LIN {X 0,Y 171.805,Z 482.478,A -85,B 0,C 180,E1 -24434.283,E2 -24434.283} C_VEL
LIN {X 0,Y 169.937,Z 475.539,A -85,B 0,C 180,E1 -24436.969,E2 -24436.969} C_VEL
LIN {X 0,Y 167.146,Z 467.963,A -85,B 0,C 180,E1 -24440.038,E2 -24440.038} C_VEL
LIN {X 0,Y 163.799,Z 461.064,A -85,B 0,C 180,E1 -24443.08,E2 -24443.08} C_VEL
LIN {X 0,Y 159.672,Z 454.191,A -85,B 0,C 180,E1 -24446.526,E2 -24446.526} C_VEL
LIN {X 0,Y 157.443,Z 450.927,A -85,B 0,C 180,E1 -24448.364,E2 -24448.364} C_VEL
LIN {X 0,Y 155.234,Z 452.338,A -85,B 0,C 180,E1 -24449.474,E2 -24449.474} C_VEL
LIN {X 0,Y 153.646,Z 452.709,A -85,B 0,C 180,E1 -24450.439,E2 -24450.439} C_VEL
LIN {X 0,Y 151.566,Z 454.907,A -85,B 0,C 180,E1 -24451.431,E2 -24451.431} C_VEL
LIN {X 0,Y 150.413,Z 455.475,A -85,B 0,C 180,E1 -24452.143,E2 -24452.143} C_VEL
LIN {X 0,Y 149.346,Z 455.04,A -85,B 0,C 180,E1 -24453.036,E2 -24453.036} C_VEL
LIN {X 0,Y 149.052,Z 454.259,A -85,B 0,C 180,E1 -24453.433,E2 -24453.433} C_VEL
LIN {X 0,Y 150.557,Z 461.284,A -85,B 0,C 180,E1 -24455.157,E2 -24455.157} C_VEL
LIN {X 0,Y 147.924,Z 476.238,A -85,B 0,C 180,E1 -24459.124,E2 -24459.124} C_VEL
LIN {X 0,Y 146.015,Z 488.722,A -85,B 0,C 180,E1 -24463.213,E2 -24463.213} C_VEL
LIN {X 0,Y 144.421,Z 500.063,A -85,B 0,C 180,E1 -24467.685,E2 -24467.685} C_VEL
LIN {X 0,Y 143.516,Z 508.412,A -85,B 0,C 180,E1 -24471.551,E2 -24471.551} C_VEL
LIN {X 0,Y 143,Z 518.672,A -85,B 0,C 180,E1 -24477.182,E2 -24477.182} C_VEL
LIN {X 0,Y 143.402,Z 525.259,A -85,B 0,C 180,E1 -24481.403,E2 -24481.403} C_VEL
LIN {X 0,Y 144.633,Z 532.666,A -85,B 0,C 180,E1 -24486.977,E2 -24486.977} C_VEL
LIN {X 0,Y 147.071,Z 538.788,A -85,B 0,C 180,E1 -24492.417,E2 -24492.417} C_VEL
LIN {X 0,Y 150.905,Z 543.761,A -85,B 0,C 180,E1 -24497.62,E2 -24497.62} C_VEL
LIN {X 0,Y 157.426,Z 548.456,A -85,B 0,C 180,E1 -24503.69,E2 -24503.69} C_VEL
LIN {X 0,Y 163.782,Z 551.125,A -85,B 0,C 180,E1 -24508.165,E2 -24508.165} C_VEL
LIN {X 0,Y 171.252,Z 552.834,A -85,B 0,C 180,E1 -24512.242,E2 -24512.242} C_VEL
LIN {X 0,Y 179.727,Z 553.572,A -85,B 0,C 180,E1 -24515.912,E2 -24515.912} C_VEL
LIN {X 0,Y 191.407,Z 553.206,A -85,B 0,C 180,E1 -24519.91,E2 -24519.91} C_VEL
LIN {X 0,Y 190.821,Z 553.718,A -85,B 0,C 180,E1 -24520.483,E2 -24520.483} C_VEL
LIN {X 0,Y 178.138,Z 559.175,A -85,B 0,C 180,E1 -24524.751,E2 -24524.751} C_VEL
LIN {X 0,Y 167.661,Z 563.079,A -85,B 0,C 180,E1 -24528.983,E2 -24528.983} C_VEL
LIN {X 0,Y 157.807,Z 566.417,A -85,B 0,C 180,E1 -24534.62,E2 -24534.62} C_VEL
LIN {X 0,Y 151.849,Z 568.111,A -85,B 0,C 180,E1 -24539.392,E2 -24539.392} C_VEL
LIN {X 0,Y 145.897,Z 569.336,A -85,B 0,C 180,E1 -24547.33,E2 -24547.33} C_VEL
LIN {X 0,Y 145.518,Z 569.56,A -85,B 0,C 180,E1 -24548.016,E2 -24548.016} C_VEL
LIN {X 0,Y 143.23,Z 574.219,A -85,B 0,C 180,E1 -24552.875,E2 -24552.875} C_VEL
LIN {X 0,Y 142.497,Z 576.289,A -85,B 0,C 180,E1 -24555.72,E2 -24555.72} C_VEL
LIN {X 0,Y 142.186,Z 579.073,A -85,B 0,C 180,E1 -24561.325,E2 -24561.325} C_VEL
LIN {X 0,Y 142.538,Z 579.938,A -85,B 0,C 180,E1 -24564.338,E2 -24564.338} C_VEL
LIN {X 0,Y 143.039,Z 580.34,A -85,B 0,C 180,E1 -24567.181,E2 -24567.181} C_VEL
LIN {X 0,Y 143.855,Z 580.307,A -85,B 0,C 180,E1 -24569.997,E2 -24569.997} C_VEL
LIN {X 0,Y 143.134,Z 579.601,A -85,B 0,C 180,E1 -24572.811,E2 -24572.811} C_VEL
LIN {X 0,Y 142.679,Z 578.492,A -85,B 0,C 180,E1 -24575.651,E2 -24575.651} C_VEL
LIN {X 0,Y 142.304,Z 576.622,A -85,B 0,C 180,E1 -24578.983,E2 -24578.983} C_VEL
LIN {X 0,Y 142.415,Z 572.404,A -85,B 0,C 180,E1 -24584.282,E2 -24584.282} C_VEL
LIN {X 0,Y 143.415,Z 567.754,A -85,B 0,C 180,E1 -24588.571,E2 -24588.571} C_VEL
LIN {X 0,Y 145.217,Z 561.884,A -85,B 0,C 180,E1 -24592.775,E2 -24592.775} C_VEL
LIN {X 0,Y 147.915,Z 554.582,A -85,B 0,C 180,E1 -24596.829,E2 -24596.829} C_VEL
LIN {X 0,Y 151.265,Z 545.507,A -85,B 0,C 180,E1 -24600.732,E2 -24600.732} C_VEL
LIN {X 0,Y 152.321,Z 541.956,A -85,B 0,C 180,E1 -24602.042,E2 -24602.042} C_VEL
LIN {X 0,Y 153.79,Z 532.793,A -85,B 0,C 180,E1 -24605.167,E2 -24605.167} C_VEL
LIN {X 0,Y 155.409,Z 522.571,A -85,B 0,C 180,E1 -24608.032,E2 -24608.032} C_VEL
LIN {X 0,Y 156.504,Z 514.859,A -85,B 0,C 180,E1 -24609.836,E2 -24609.836} C_VEL
LIN {X 0,Y 156.689,Z 509.881,A -85,B 0,C 180,E1 -24610.999,E2 -24610.999} C_VEL
LIN {X 0,Y 155.545,Z 501.863,A -85,B 0,C 180,E1 -24613.085,E2 -24613.085} C_VEL
LIN {X 0,Y 154.315,Z 495.338,A -85,B 0,C 180,E1 -24614.705,E2 -24614.705} C_VEL
LIN {X 0,Y 153.628,Z 488.352,A -85,B 0,C 180,E1 -24616.066,E2 -24616.066} C_VEL
LIN {X 0,Y 152.596,Z 475.837,A -85,B 0,C 180,E1 -24618.1,E2 -24618.1} C_VEL
LIN {X 0,Y 151.177,Z 468.093,A -85,B 0,C 180,E1 -24619.396,E2 -24619.396} C_VEL
LIN {X 0,Y 145.37,Z 455.802,A -85,B 0,C 180,E1 -24622.894,E2 -24622.894} C_VEL
LIN {X 0,Y 144.25,Z 450.728,A -85,B 0,C 180,E1 -24625.337,E2 -24625.337} C_VEL
LIN {X 0,Y 142.137,Z 443.856,A -85,B 0,C 180,E1 -24629.227,E2 -24629.227} C_VEL
LIN {X 0,Y 140.598,Z 440.661,A -85,B 0,C 180,E1 -24631.65,E2 -24631.65} C_VEL
LIN {X 0,Y 139.499,Z 439.298,A -85,B 0,C 180,E1 -24633.037,E2 -24633.037} C_VEL
LIN {X 0,Y 137.889,Z 436.001,A -85,B 0,C 180,E1 -24635.937,E2 -24635.937} C_VEL
LIN {X 0,Y 136.434,Z 433.163,A -85,B 0,C 180,E1 -24638.865,E2 -24638.865} C_VEL
LIN {X 0,Y 136.27,Z 432.124,A -85,B 0,C 180,E1 -24639.825,E2 -24639.825} C_VEL
LIN {X 0,Y 136.489,Z 432.104,A -85,B 0,C 180,E1 -24648.115,E2 -24648.115} C_VEL
LIN {X 0,Y 136.58,Z 432.088,A -85,B 0,C 180,E1 -24651.12,E2 -24651.12} C_VEL
LIN {X 0,Y 137.127,Z 432.018,A -85,B 0,C 180,E1 -24660.001,E2 -24660.001} C_VEL
LIN {X 0,Y 136.571,Z 432.045,A -85,B 0,C 180,E1 -24668.882,E2 -24668.882} C_VEL
LIN {X 0,Y 136.483,Z 432.078,A -85,B 0,C 180,E1 -24671.956,E2 -24671.956} C_VEL
LIN {X 0,Y 136.244,Z 432.129,A -85,B 0,C 180,E1 -24678.03,E2 -24678.03} C_VEL
LIN {X 0,Y 136.191,Z 432.134,A -85,B 0,C 180,E1 -24681.751,E2 -24681.751} C_VEL
LIN {X 0,Y 136.093,Z 432.113,A -85,B 0,C 180,E1 -24688.618,E2 -24688.618} C_VEL
LIN {X 0,Y 136.142,Z 432.245,A -85,B 0,C 180,E1 -24692.385,E2 -24692.385} C_VEL
LIN {X 0,Y 137.183,Z 435.226,A -85,B 0,C 180,E1 -24695.757,E2 -24695.757} C_VEL
LIN {X 0,Y 141.142,Z 440.004,A -85,B 0,C 180,E1 -24698.55,E2 -24698.55} C_VEL
LIN {X 0,Y 144.042,Z 443.761,A -85,B 0,C 180,E1 -24700.508,E2 -24700.508} C_VEL
LIN {X 0,Y 146.952,Z 448.113,A -85,B 0,C 180,E1 -24702.496,E2 -24702.496} C_VEL
LIN {X 0,Y 150.969,Z 454.759,A -85,B 0,C 180,E1 -24705.307,E2 -24705.307} C_VEL
LIN {X 0,Y 155.269,Z 463.772,A -85,B 0,C 180,E1 -24708.703,E2 -24708.703} C_VEL
LIN {X 0,Y 158.22,Z 471.79,A -85,B 0,C 180,E1 -24711.551,E2 -24711.551} C_VEL
LIN {X 0,Y 160.626,Z 481.017,A -85,B 0,C 180,E1 -24714.765,E2 -24714.765} C_VEL
LIN {X 0,Y 160.992,Z 482.859,A -85,B 0,C 180,E1 -24715.427,E2 -24715.427} C_VEL
LIN {X 0,Y 160.557,Z 485.505,A -85,B 0,C 180,E1 -24716.08,E2 -24716.08} C_VEL
LIN {X 0,Y 156.85,Z 496.328,A -85,B 0,C 180,E1 -24718.75,E2 -24718.75} C_VEL
LIN {X 0,Y 152.896,Z 506.216,A -85,B 0,C 180,E1 -24721.895,E2 -24721.895} C_VEL
LIN {X 0,Y 148.976,Z 515.07,A -85,B 0,C 180,E1 -24725.624,E2 -24725.624} C_VEL
LIN {X 0,Y 145.507,Z 522.195,A -85,B 0,C 180,E1 -24729.505,E2 -24729.505} C_VEL
LIN {X 0,Y 143.222,Z 526.998,A -85,B 0,C 180,E1 -24732.88,E2 -24732.88} C_VEL
LIN {X 0,Y 140.788,Z 531.675,A -85,B 0,C 180,E1 -24737.022,E2 -24737.022} C_VEL
LIN {X 0,Y 138.855,Z 535.27,A -85,B 0,C 180,E1 -24741.27,E2 -24741.27} C_VEL
LIN {X 0,Y 137.973,Z 537.117,A -85,B 0,C 180,E1 -24744.156,E2 -24744.156} C_VEL
LIN {X 0,Y 137.419,Z 538.522,A -85,B 0,C 180,E1 -24747.072,E2 -24747.072} C_VEL
LIN {X 0,Y 137.226,Z 540.113,A -85,B 0,C 180,E1 -24752.939,E2 -24752.939} C_VEL
LIN {X 0,Y 137.317,Z 540.381,A -85,B 0,C 180,E1 -24755.878,E2 -24755.878} C_VEL
LIN {X 0,Y 137.608,Z 540.235,A -85,B 0,C 180,E1 -24758.817,E2 -24758.817} C_VEL
LIN {X 0,Y 139.808,Z 538.683,A -85,B 0,C 180,E1 -24764.56,E2 -24764.56} C_VEL
LIN {X 0,Y 141.286,Z 537.324,A -85,B 0,C 180,E1 -24767.368,E2 -24767.368} C_VEL
LIN {X 0,Y 143.838,Z 534.273,A -85,B 0,C 180,E1 -24771.819,E2 -24771.819} C_VEL
LIN {X 0,Y 147.707,Z 529.137,A -85,B 0,C 180,E1 -24776.876,E2 -24776.876} C_VEL
LIN {X 0,Y 151.298,Z 523.764,A -85,B 0,C 180,E1 -24780.731,E2 -24780.731} C_VEL
LIN {X 0,Y 155.503,Z 516.959,A -85,B 0,C 180,E1 -24784.401,E2 -24784.401} C_VEL
LIN {X 0,Y 160.227,Z 508.406,A -85,B 0,C 180,E1 -24787.888,E2 -24787.888} C_VEL
LIN {X 0,Y 164.531,Z 499.594,A -85,B 0,C 180,E1 -24790.651,E2 -24790.651} C_VEL
LIN {X 0,Y 167.149,Z 493.293,A -85,B 0,C 180,E1 -24792.282,E2 -24792.282} C_VEL
LIN {X 0,Y 166.758,Z 488.389,A -85,B 0,C 180,E1 -24794.236,E2 -24794.236} C_VEL
LIN {X 0,Y 164.998,Z 480.301,A -85,B 0,C 180,E1 -24797.615,E2 -24797.615} C_VEL
LIN {X 0,Y 162.856,Z 473.543,A -85,B 0,C 180,E1 -24800.545,E2 -24800.545} C_VEL
LIN {X 0,Y 159.432,Z 465.725,A -85,B 0,C 180,E1 -24804.261,E2 -24804.261} C_VEL
LIN {X 0,Y 155.545,Z 458.948,A -85,B 0,C 180,E1 -24807.987,E2 -24807.987} C_VEL
LIN {X 0,Y 154.773,Z 458.892,A -85,B 0,C 180,E1 -24808.475,E2 -24808.475} C_VEL
LIN {X 0,Y 153.201,Z 459.625,A -85,B 0,C 180,E1 -24809.312,E2 -24809.312} C_VEL
LIN {X 0,Y 150.645,Z 461.659,A -85,B 0,C 180,E1 -24810.559,E2 -24810.559} C_VEL
LIN {X 0,Y 148.706,Z 462.303,A -85,B 0,C 180,E1 -24811.795,E2 -24811.795} C_VEL
LIN {X 0,Y 144.741,Z 465.331,A -85,B 0,C 180,E1 -24814.086,E2 -24814.086} C_VEL
LIN {X 0,Y 143.085,Z 466.026,A -85,B 0,C 180,E1 -24815.322,E2 -24815.322} C_VEL
LIN {X 0,Y 142.719,Z 465.473,A -85,B 0,C 180,E1 -24815.932,E2 -24815.932} C_VEL
LIN {X 0,Y 140.372,Z 478.948,A -85,B 0,C 180,E1 -24819.866,E2 -24819.866} C_VEL
LIN {X 0,Y 138.522,Z 491.22,A -85,B 0,C 180,E1 -24824.213,E2 -24824.213} C_VEL
LIN {X 0,Y 136.942,Z 503.88,A -85,B 0,C 180,E1 -24829.651,E2 -24829.651} C_VEL
LIN {X 0,Y 135.988,Z 515.026,A -85,B 0,C 180,E1 -24835.553,E2 -24835.553} C_VEL
LIN {X 0,Y 136.288,Z 523.292,A -85,B 0,C 180,E1 -24840.738,E2 -24840.738} C_VEL
LIN {X 0,Y 137.599,Z 532.127,A -85,B 0,C 180,E1 -24847.335,E2 -24847.335} C_VEL
LIN {X 0,Y 140.151,Z 538.583,A -85,B 0,C 180,E1 -24853.041,E2 -24853.041} C_VEL
LIN {X 0,Y 145.344,Z 545.059,A -85,B 0,C 180,E1 -24859.784,E2 -24859.784} C_VEL
LIN {X 0,Y 150.972,Z 549.028,A -85,B 0,C 180,E1 -24864.769,E2 -24864.769} C_VEL
LIN {X 0,Y 157.609,Z 552.021,A -85,B 0,C 180,E1 -24869.373,E2 -24869.373} C_VEL
LIN {X 0,Y 165.381,Z 554.072,A -85,B 0,C 180,E1 -24873.534,E2 -24873.534} C_VEL
LIN {X 0,Y 174.177,Z 555.197,A -85,B 0,C 180,E1 -24877.246,E2 -24877.246} C_VEL
LIN {X 0,Y 181.439,Z 555.419,A -85,B 0,C 180,E1 -24879.775,E2 -24879.775} C_VEL
LIN {X 0,Y 180.961,Z 555.879,A -85,B 0,C 180,E1 -24880.385,E2 -24880.385} C_VEL
LIN {X 0,Y 168.483,Z 560.407,A -85,B 0,C 180,E1 -24884.833,E2 -24884.833} C_VEL
LIN {X 0,Y 159.674,Z 563.108,A -85,B 0,C 180,E1 -24888.68,E2 -24888.68} C_VEL
LIN {X 0,Y 152.091,Z 565.208,A -85,B 0,C 180,E1 -24893.075,E2 -24893.075} C_VEL
LIN {X 0,Y 143.319,Z 567.038,A -85,B 0,C 180,E1 -24900.632,E2 -24900.632} C_VEL
LIN {X 0,Y 139.662,Z 567.468,A -85,B 0,C 180,E1 -24905.885,E2 -24905.885} C_VEL
LIN {X 0,Y 136.991,Z 572.091,A -85,B 0,C 180,E1 -24910.518,E2 -24910.518} C_VEL
LIN {X 0,Y 135.568,Z 575.311,A -85,B 0,C 180,E1 -24914.974,E2 -24914.974} C_VEL
LIN {X 0,Y 135.12,Z 576.919,A -85,B 0,C 180,E1 -24917.989,E2 -24917.989} C_VEL
LIN {X 0,Y 135.45,Z 578.932,A -85,B 0,C 180,E1 -24924.04,E2 -24924.04} C_VEL
LIN {X 0,Y 135.939,Z 579.326,A -85,B 0,C 180,E1 -24927.033,E2 -24927.033} C_VEL
LIN {X 0,Y 136.764,Z 579.281,A -85,B 0,C 180,E1 -24929.997,E2 -24929.997} C_VEL
LIN {X 0,Y 136.03,Z 578.564,A -85,B 0,C 180,E1 -24932.958,E2 -24932.958} C_VEL
LIN {X 0,Y 135.579,Z 577.444,A -85,B 0,C 180,E1 -24935.947,E2 -24935.947} C_VEL
LIN {X 0,Y 135.24,Z 575.771,A -85,B 0,C 180,E1 -24939.118,E2 -24939.118} C_VEL
LIN {X 0,Y 135.425,Z 571.309,A -85,B 0,C 180,E1 -24945.036,E2 -24945.036} C_VEL
LIN {X 0,Y 136.585,Z 566.64,A -85,B 0,C 180,E1 -24949.536,E2 -24949.536} C_VEL
LIN {X 0,Y 138.827,Z 560.132,A -85,B 0,C 180,E1 -24954.325,E2 -24954.325} C_VEL
LIN {X 0,Y 142.076,Z 552.029,A -85,B 0,C 180,E1 -24958.832,E2 -24958.832} C_VEL
LIN {X 0,Y 145.122,Z 544.318,A -85,B 0,C 180,E1 -24962.185,E2 -24962.185} C_VEL
LIN {X 0,Y 147.098,Z 534.44,A -85,B 0,C 180,E1 -24965.904,E2 -24965.904} C_VEL
LIN {X 0,Y 149.05,Z 523.917,A -85,B 0,C 180,E1 -24969.094,E2 -24969.094} C_VEL
LIN {X 0,Y 150.937,Z 512.662,A -85,B 0,C 180,E1 -24971.842,E2 -24971.842} C_VEL
LIN {X 0,Y 152.621,Z 501.143,A -85,B 0,C 180,E1 -24974.056,E2 -24974.056} C_VEL
LIN {X 0,Y 153.683,Z 490.333,A -85,B 0,C 180,E1 -24975.732,E2 -24975.732} C_VEL
LIN {X 0,Y 153.628,Z 488.352,A -85,B 0,C 180,E1 -24976.066,E2 -24976.066} C_VEL
LIN {X 0,Y 152.956,Z 483.098,A -85,B 0,C 180,E1 -24977.077,E2 -24977.077} C_VEL
LIN {X 0,Y 150.674,Z 476.845,A -85,B 0,C 180,E1 -24978.733,E2 -24978.733} C_VEL
LIN {X 0,Y 146.728,Z 469.819,A -85,B 0,C 180,E1 -24981.137,E2 -24981.137} C_VEL
LIN {X 0,Y 143.421,Z 464.323,A -85,B 0,C 180,E1 -24983.156,E2 -24983.156} C_VEL
LIN {X 0,Y 138.725,Z 454.306,A -85,B 0,C 180,E1 -24986.569,E2 -24986.569} C_VEL
LIN {X 0,Y 137.507,Z 449.61,A -85,B 0,C 180,E1 -24989.264,E2 -24989.264} C_VEL
LIN {X 0,Y 135.708,Z 445.682,A -85,B 0,C 180,E1 -24992.22,E2 -24992.22} C_VEL
LIN {X 0,Y 131.769,Z 438.096,A -85,B 0,C 180,E1 -24999.716,E2 -24999.716} C_VEL
LIN {X 0,Y 129.406,Z 433.796,A -85,B 0,C 180,E1 -25005.855,E2 -25005.855} C_VEL
LIN {X 0,Y 129.333,Z 432.999,A -85,B 0,C 180,E1 -25007.048,E2 -25007.048} C_VEL
LIN {X 0,Y 129.506,Z 432.966,A -85,B 0,C 180,E1 -25010.631,E2 -25010.631} C_VEL
LIN {X 0,Y 130.082,Z 432.895,A -85,B 0,C 180,E1 -25020.001,E2 -25020.001} C_VEL
LIN {X 0,Y 129.5,Z 432.924,A -85,B 0,C 180,E1 -25029.371,E2 -25029.371} C_VEL
LIN {X 0,Y 129.386,Z 432.969,A -85,B 0,C 180,E1 -25032.55,E2 -25032.55} C_VEL
LIN {X 0,Y 129.153,Z 433.019,A -85,B 0,C 180,E1 -25039.057,E2 -25039.057} C_VEL
LIN {X 0,Y 129.013,Z 433.04,A -85,B 0,C 180,E1 -25044.973,E2 -25044.973} C_VEL
LIN {X 0,Y 129.044,Z 433.273,A -85,B 0,C 180,E1 -25045.831,E2 -25045.831} C_VEL
LIN {X 0,Y 130.673,Z 436.736,A -85,B 0,C 180,E1 -25051.288,E2 -25051.288} C_VEL
LIN {X 0,Y 136.497,Z 443.699,A -85,B 0,C 180,E1 -25056.194,E2 -25056.194} C_VEL
LIN {X 0,Y 140.572,Z 449.281,A -85,B 0,C 180,E1 -25059.371,E2 -25059.371} C_VEL
LIN {X 0,Y 145.033,Z 456.594,A -85,B 0,C 180,E1 -25062.916,E2 -25062.916} C_VEL
LIN {X 0,Y 149.652,Z 466.342,A -85,B 0,C 180,E1 -25067.014,E2 -25067.014} C_VEL
LIN {X 0,Y 152.721,Z 475.183,A -85,B 0,C 180,E1 -25070.428,E2 -25070.428} C_VEL
LIN {X 0,Y 154.852,Z 484.253,A -85,B 0,C 180,E1 -25073.846,E2 -25073.846} C_VEL
LIN {X 0,Y 155.065,Z 485.477,A -85,B 0,C 180,E1 -25074.305,E2 -25074.305} C_VEL
LIN {X 0,Y 151.601,Z 495.729,A -85,B 0,C 180,E1 -25076.838,E2 -25076.838} C_VEL
LIN {X 0,Y 147.528,Z 505.678,A -85,B 0,C 180,E1 -25079.99,E2 -25079.99} C_VEL
LIN {X 0,Y 143.224,Z 514.916,A -85,B 0,C 180,E1 -25083.796,E2 -25083.796} C_VEL
LIN {X 0,Y 139.531,Z 522.236,A -85,B 0,C 180,E1 -25087.808,E2 -25087.808} C_VEL
LIN {X 0,Y 136.539,Z 528.097,A -85,B 0,C 180,E1 -25092.015,E2 -25092.015} C_VEL
LIN {X 0,Y 133.953,Z 532.756,A -85,B 0,C 180,E1 -25096.347,E2 -25096.347} C_VEL
LIN {X 0,Y 131.917,Z 536.331,A -85,B 0,C 180,E1 -25100.807,E2 -25100.807} C_VEL
LIN {X 0,Y 130.987,Z 538.169,A -85,B 0,C 180,E1 -25103.843,E2 -25103.843} C_VEL
LIN {X 0,Y 130.402,Z 539.557,A -85,B 0,C 180,E1 -25106.914,E2 -25106.914} C_VEL
LIN {X 0,Y 130.206,Z 541.131,A -85,B 0,C 180,E1 -25113.097,E2 -25113.097} C_VEL
LIN {X 0,Y 130.324,Z 541.387,A -85,B 0,C 180,E1 -25116.195,E2 -25116.195} C_VEL
LIN {X 0,Y 130.661,Z 541.227,A -85,B 0,C 180,E1 -25119.289,E2 -25119.289} C_VEL
LIN {X 0,Y 133.016,Z 539.656,A -85,B 0,C 180,E1 -25125.321,E2 -25125.321} C_VEL
LIN {X 0,Y 134.591,Z 538.281,A -85,B 0,C 180,E1 -25128.262,E2 -25128.262} C_VEL
LIN {X 0,Y 137.314,Z 535.23,A -85,B 0,C 180,E1 -25132.884,E2 -25132.884} C_VEL
LIN {X 0,Y 141.464,Z 530.053,A -85,B 0,C 180,E1 -25138.165,E2 -25138.165} C_VEL
LIN {X 0,Y 145.292,Z 524.656,A -85,B 0,C 180,E1 -25142.15,E2 -25142.15} C_VEL
LIN {X 0,Y 149.739,Z 517.814,A -85,B 0,C 180,E1 -25145.925,E2 -25145.925} C_VEL
LIN {X 0,Y 154.739,Z 509.226,A -85,B 0,C 180,E1 -25149.487,E2 -25149.487} C_VEL
LIN {X 0,Y 159.252,Z 500.377,A -85,B 0,C 180,E1 -25152.302,E2 -25152.302} C_VEL
LIN {X 0,Y 161.44,Z 495.179,A -85,B 0,C 180,E1 -25153.72,E2 -25153.72} C_VEL
LIN {X 0,Y 160.715,Z 489.007,A -85,B 0,C 180,E1 -25156.469,E2 -25156.469} C_VEL
LIN {X 0,Y 159.299,Z 482.369,A -85,B 0,C 180,E1 -25159.484,E2 -25159.484} C_VEL
LIN {X 0,Y 156.998,Z 475.117,A -85,B 0,C 180,E1 -25162.98,E2 -25162.98} C_VEL
LIN {X 0,Y 154.432,Z 469.217,A -85,B 0,C 180,E1 -25166.117,E2 -25166.117} C_VEL
LIN {X 0,Y 152.726,Z 466,A -85,B 0,C 180,E1 -25168.048,E2 -25168.048} C_VEL
LIN {X 0,Y 150.464,Z 467.627,A -85,B 0,C 180,E1 -25169.082,E2 -25169.082} C_VEL
LIN {X 0,Y 146.504,Z 469.484,A -85,B 0,C 180,E1 -25171.332,E2 -25171.332} C_VEL
LIN {X 0,Y 144.368,Z 471.091,A -85,B 0,C 180,E1 -25172.452,E2 -25172.452} C_VEL
LIN {X 0,Y 142.493,Z 472.128,A -85,B 0,C 180,E1 -25173.646,E2 -25173.646} C_VEL
LIN {X 0,Y 140.43,Z 473.854,A -85,B 0,C 180,E1 -25174.825,E2 -25174.825} C_VEL
LIN {X 0,Y 136.879,Z 477.797,A -85,B 0,C 180,E1 -25176.551,E2 -25176.551} C_VEL
LIN {X 0,Y 135.859,Z 478.73,A -85,B 0,C 180,E1 -25177.171,E2 -25177.171} C_VEL
LIN {X 0,Y 134.15,Z 479.926,A -85,B 0,C 180,E1 -25178.485,E2 -25178.485} C_VEL
LIN {X 0,Y 133.163,Z 479.611,A -85,B 0,C 180,E1 -25180.037,E2 -25180.037} C_VEL
LIN {X 0,Y 131.339,Z 491.547,A -85,B 0,C 180,E1 -25184.48,E2 -25184.48} C_VEL
LIN {X 0,Y 129.85,Z 503.51,A -85,B 0,C 180,E1 -25189.868,E2 -25189.868} C_VEL
LIN {X 0,Y 128.926,Z 514.916,A -85,B 0,C 180,E1 -25196.092,E2 -25196.092} C_VEL
LIN {X 0,Y 129.318,Z 523.345,A -85,B 0,C 180,E1 -25201.556,E2 -25201.556} C_VEL
LIN {X 0,Y 130.607,Z 531.449,A -85,B 0,C 180,E1 -25207.73,E2 -25207.73} C_VEL
LIN {X 0,Y 133.254,Z 538.245,A -85,B 0,C 180,E1 -25213.729,E2 -25213.729} C_VEL
LIN {X 0,Y 137.462,Z 543.88,A -85,B 0,C 180,E1 -25219.409,E2 -25219.409} C_VEL
LIN {X 0,Y 144.565,Z 549.414,A -85,B 0,C 180,E1 -25225.946,E2 -25225.946} C_VEL
LIN {X 0,Y 151.513,Z 552.792,A -85,B 0,C 180,E1 -25230.679,E2 -25230.679} C_VEL
LIN {X 0,Y 159.592,Z 555.197,A -85,B 0,C 180,E1 -25234.923,E2 -25234.923} C_VEL
LIN {X 0,Y 170.706,Z 556.893,A -85,B 0,C 180,E1 -25239.38,E2 -25239.38} C_VEL
LIN {X 0,Y 171.241,Z 557.378,A -85,B 0,C 180,E1 -25240.306,E2 -25240.306} C_VEL
LIN {X 0,Y 158.865,Z 560.943,A -85,B 0,C 180,E1 -25244.939,E2 -25244.939} C_VEL
LIN {X 0,Y 150.328,Z 563.031,A -85,B 0,C 180,E1 -25249.114,E2 -25249.114} C_VEL
LIN {X 0,Y 139.976,Z 564.935,A -85,B 0,C 180,E1 -25256.472,E2 -25256.472} C_VEL
LIN {X 0,Y 133.887,Z 565.494,A -85,B 0,C 180,E1 -25263.744,E2 -25263.744} C_VEL
LIN {X 0,Y 131.038,Z 569.819,A -85,B 0,C 180,E1 -25267.946,E2 -25267.946} C_VEL
LIN {X 0,Y 129.082,Z 573.353,A -85,B 0,C 180,E1 -25272.572,E2 -25272.572} C_VEL
LIN {X 0,Y 128.121,Z 575.923,A -85,B 0,C 180,E1 -25277.322,E2 -25277.322} C_VEL
LIN {X 0,Y 128.359,Z 577.925,A -85,B 0,C 180,E1 -25283.71,E2 -25283.71} C_VEL
LIN {X 0,Y 128.838,Z 578.31,A -85,B 0,C 180,E1 -25286.87,E2 -25286.87} C_VEL
LIN {X 0,Y 129.676,Z 578.256,A -85,B 0,C 180,E1 -25289.997,E2 -25289.997} C_VEL
LIN {X 0,Y 128.927,Z 577.527,A -85,B 0,C 180,E1 -25293.121,E2 -25293.121} C_VEL
LIN {X 0,Y 128.463,Z 576.393,A -85,B 0,C 180,E1 -25296.278,E2 -25296.278} C_VEL
LIN {X 0,Y 128.082,Z 573.815,A -85,B 0,C 180,E1 -25301.069,E2 -25301.069} C_VEL
LIN {X 0,Y 128.474,Z 570.216,A -85,B 0,C 180,E1 -25305.87,E2 -25305.87} C_VEL
LIN {X 0,Y 129.811,Z 565.529,A -85,B 0,C 180,E1 -25310.6,E2 -25310.6} C_VEL
LIN {X 0,Y 132.512,Z 558.474,A -85,B 0,C 180,E1 -25315.944,E2 -25315.944} C_VEL
LIN {X 0,Y 135.806,Z 550.865,A -85,B 0,C 180,E1 -25320.298,E2 -25320.298} C_VEL
LIN {X 0,Y 138.886,Z 543.09,A -85,B 0,C 180,E1 -25323.819,E2 -25323.819} C_VEL
LIN {X 0,Y 140.987,Z 533.364,A -85,B 0,C 180,E1 -25327.632,E2 -25327.632} C_VEL
LIN {X 0,Y 143.273,Z 522.572,A -85,B 0,C 180,E1 -25330.997,E2 -25330.997} C_VEL
LIN {X 0,Y 145.434,Z 511.097,A -85,B 0,C 180,E1 -25333.861,E2 -25333.861} C_VEL
LIN {X 0,Y 147.465,Z 498.539,A -85,B 0,C 180,E1 -25336.28,E2 -25336.28} C_VEL
LIN {X 0,Y 148.217,Z 491.08,A -85,B 0,C 180,E1 -25337.493,E2 -25337.493} C_VEL
LIN {X 0,Y 147.659,Z 479.337,A -85,B 0,C 180,E1 -25339.595,E2 -25339.595} C_VEL
LIN {X 0,Y 146.686,Z 471.856,A -85,B 0,C 180,E1 -25340.931,E2 -25340.931} C_VEL
LIN {X 0,Y 143.421,Z 464.323,A -85,B 0,C 180,E1 -25343.156,E2 -25343.156} C_VEL
LIN {X 0,Y 140.911,Z 460.619,A -85,B 0,C 180,E1 -25344.732,E2 -25344.732} C_VEL
LIN {X 0,Y 136.291,Z 455.849,A -85,B 0,C 180,E1 -25347.787,E2 -25347.787} C_VEL
LIN {X 0,Y 131.421,Z 451.317,A -85,B 0,C 180,E1 -25352.093,E2 -25352.093} C_VEL
LIN {X 0,Y 130.236,Z 449.835,A -85,B 0,C 180,E1 -25353.644,E2 -25353.644} C_VEL
LIN {X 0,Y 126.937,Z 443.072,A -85,B 0,C 180,E1 -25360.599,E2 -25360.599} C_VEL
LIN {X 0,Y 124.67,Z 438.557,A -85,B 0,C 180,E1 -25366.969,E2 -25366.969} C_VEL
LIN {X 0,Y 122.838,Z 433.805,A -85,B 0,C 180,E1 -25378.771,E2 -25378.771} C_VEL
LIN {X 0,Y 123.036,Z 433.772,A -85,B 0,C 180,E1 -25380.001,E2 -25380.001} C_VEL
LIN {X 0,Y 122.404,Z 433.814,A -85,B 0,C 180,E1 -25387.137,E2 -25387.137} C_VEL
LIN {X 0,Y 122.355,Z 433.84,A -85,B 0,C 180,E1 -25392.473,E2 -25392.473} C_VEL
LIN {X 0,Y 122.802,Z 436.27,A -85,B 0,C 180,E1 -25400.084,E2 -25400.084} C_VEL
LIN {X 0,Y 124.245,Z 438.461,A -85,B 0,C 180,E1 -25405.581,E2 -25405.581} C_VEL
LIN {X 0,Y 127.692,Z 442.456,A -85,B 0,C 180,E1 -25409.467,E2 -25409.467} C_VEL
LIN {X 0,Y 129.418,Z 444.245,A -85,B 0,C 180,E1 -25411.175,E2 -25411.175} C_VEL
LIN {X 0,Y 133.877,Z 450.1,A -85,B 0,C 180,E1 -25415.388,E2 -25415.388} C_VEL
LIN {X 0,Y 137.193,Z 455.092,A -85,B 0,C 180,E1 -25418.4,E2 -25418.4} C_VEL
LIN {X 0,Y 140.314,Z 460.669,A -85,B 0,C 180,E1 -25421.301,E2 -25421.301} C_VEL
LIN {X 0,Y 143.701,Z 467.997,A -85,B 0,C 180,E1 -25424.743,E2 -25424.743} C_VEL
LIN {X 0,Y 146.466,Z 475.686,A -85,B 0,C 180,E1 -25428.051,E2 -25428.051} C_VEL
LIN {X 0,Y 148.475,Z 484.061,A -85,B 0,C 180,E1 -25431.455,E2 -25431.455} C_VEL
LIN {X 0,Y 149.139,Z 488.055,A -85,B 0,C 180,E1 -25433.076,E2 -25433.076} C_VEL
LIN {X 0,Y 145.198,Z 498.43,A -85,B 0,C 180,E1 -25435.775,E2 -25435.775} C_VEL
LIN {X 0,Y 140.682,Z 508.587,A -85,B 0,C 180,E1 -25439.203,E2 -25439.203} C_VEL
LIN {X 0,Y 136.333,Z 517.361,A -85,B 0,C 180,E1 -25443.192,E2 -25443.192} C_VEL
LIN {X 0,Y 132.503,Z 524.431,A -85,B 0,C 180,E1 -25447.388,E2 -25447.388} C_VEL
LIN {X 0,Y 129.889,Z 529.196,A -85,B 0,C 180,E1 -25451.06,E2 -25451.06} C_VEL
LIN {X 0,Y 127.166,Z 533.832,A -85,B 0,C 180,E1 -25455.603,E2 -25455.603} C_VEL
LIN {X 0,Y 124.988,Z 537.392,A -85,B 0,C 180,E1 -25460.292,E2 -25460.292} C_VEL
LIN {X 0,Y 124.006,Z 539.221,A -85,B 0,C 180,E1 -25463.495,E2 -25463.495} C_VEL
LIN {X 0,Y 123.387,Z 540.591,A -85,B 0,C 180,E1 -25466.738,E2 -25466.738} C_VEL
LIN {X 0,Y 123.188,Z 542.148,A -85,B 0,C 180,E1 -25473.274,E2 -25473.274} C_VEL
LIN {X 0,Y 123.336,Z 542.391,A -85,B 0,C 180,E1 -25476.547,E2 -25476.547} C_VEL
LIN {X 0,Y 123.724,Z 542.219,A -85,B 0,C 180,E1 -25479.815,E2 -25479.815} C_VEL
LIN {X 0,Y 126.249,Z 540.63,A -85,B 0,C 180,E1 -25486.164,E2 -25486.164} C_VEL
LIN {X 0,Y 127.932,Z 539.236,A -85,B 0,C 180,E1 -25489.249,E2 -25489.249} C_VEL
LIN {X 0,Y 130.853,Z 536.178,A -85,B 0,C 180,E1 -25494.067,E2 -25494.067} C_VEL
LIN {X 0,Y 134.052,Z 532.513,A -85,B 0,C 180,E1 -25498.158,E2 -25498.158} C_VEL
LIN {X 0,Y 137.925,Z 527.488,A -85,B 0,C 180,E1 -25502.349,E2 -25502.349} C_VEL
LIN {X 0,Y 142.511,Z 521.112,A -85,B 0,C 180,E1 -25506.287,E2 -25506.287} C_VEL
LIN {X 0,Y 146.802,Z 514.365,A -85,B 0,C 180,E1 -25509.518,E2 -25509.518} C_VEL
LIN {X 0,Y 151.267,Z 506.685,A -85,B 0,C 180,E1 -25512.355,E2 -25512.355} C_VEL
LIN {X 0,Y 155.502,Z 498.111,A -85,B 0,C 180,E1 -25514.91,E2 -25514.91} C_VEL
LIN {X 0,Y 155.678,Z 496.464,A -85,B 0,C 180,E1 -25515.595,E2 -25515.595} C_VEL
LIN {X 0,Y 154.577,Z 488.204,A -85,B 0,C 180,E1 -25519.616,E2 -25519.616} C_VEL
LIN {X 0,Y 152.784,Z 481.093,A -85,B 0,C 180,E1 -25523.273,E2 -25523.273} C_VEL
LIN {X 0,Y 150.388,Z 474.599,A -85,B 0,C 180,E1 -25526.935,E2 -25526.935} C_VEL
LIN {X 0,Y 149.941,Z 473.671,A -85,B 0,C 180,E1 -25527.536,E2 -25527.536} C_VEL
LIN {X 0,Y 146.01,Z 475.351,A -85,B 0,C 180,E1 -25529.641,E2 -25529.641} C_VEL
LIN {X 0,Y 141.786,Z 477.908,A -85,B 0,C 180,E1 -25531.907,E2 -25531.907} C_VEL
LIN {X 0,Y 139.562,Z 479.673,A -85,B 0,C 180,E1 -25533.049,E2 -25533.049} C_VEL
LIN {X 0,Y 135.809,Z 483.289,A -85,B 0,C 180,E1 -25534.733,E2 -25534.733} C_VEL
LIN {X 0,Y 134.715,Z 484.217,A -85,B 0,C 180,E1 -25535.331,E2 -25535.331} C_VEL
LIN {X 0,Y 132.835,Z 485.492,A -85,B 0,C 180,E1 -25536.62,E2 -25536.62} C_VEL
LIN {X 0,Y 131.244,Z 486.298,A -85,B 0,C 180,E1 -25537.984,E2 -25537.984} C_VEL
LIN {X 0,Y 129.392,Z 487.778,A -85,B 0,C 180,E1 -25539.325,E2 -25539.325} C_VEL
LIN {X 0,Y 127.323,Z 489.737,A -85,B 0,C 180,E1 -25540.658,E2 -25540.658} C_VEL
LIN {X 0,Y 125.364,Z 491.284,A -85,B 0,C 180,E1 -25542.379,E2 -25542.379} C_VEL
LIN {X 0,Y 124.275,Z 491.532,A -85,B 0,C 180,E1 -25544.156,E2 -25544.156} C_VEL
LIN {X 0,Y 124.213,Z 491.312,A -85,B 0,C 180,E1 -25544.595,E2 -25544.595} C_VEL
LIN {X 0,Y 122.753,Z 503.048,A -85,B 0,C 180,E1 -25550.109,E2 -25550.109} C_VEL
LIN {X 0,Y 121.933,Z 513.288,A -85,B 0,C 180,E1 -25555.868,E2 -25555.868} C_VEL
LIN {X 0,Y 122.308,Z 522.085,A -85,B 0,C 180,E1 -25561.646,E2 -25561.646} C_VEL
LIN {X 0,Y 123.623,Z 530.548,A -85,B 0,C 180,E1 -25568.17,E2 -25568.17} C_VEL
LIN {X 0,Y 126.384,Z 537.68,A -85,B 0,C 180,E1 -25574.491,E2 -25574.491} C_VEL
LIN {X 0,Y 132.082,Z 544.995,A -85,B 0,C 180,E1 -25581.867,E2 -25581.867} C_VEL
LIN {X 0,Y 138.218,Z 549.642,A -85,B 0,C 180,E1 -25587.233,E2 -25587.233} C_VEL
LIN {X 0,Y 145.483,Z 553.345,A -85,B 0,C 180,E1 -25592.099,E2 -25592.099} C_VEL
LIN {X 0,Y 153.886,Z 556.157,A -85,B 0,C 180,E1 -25596.42,E2 -25596.42} C_VEL
LIN {X 0,Y 161.63,Z 557.746,A -85,B 0,C 180,E1 -25599.579,E2 -25599.579} C_VEL
LIN {X 0,Y 160.591,Z 558.362,A -85,B 0,C 180,E1 -25600.569,E2 -25600.569} C_VEL
LIN {X 0,Y 149.354,Z 560.838,A -85,B 0,C 180,E1 -25605.099,E2 -25605.099} C_VEL
LIN {X 0,Y 137.483,Z 562.787,A -85,B 0,C 180,E1 -25612.159,E2 -25612.159} C_VEL
LIN {X 0,Y 131.355,Z 563.304,A -85,B 0,C 180,E1 -25617.65,E2 -25617.65} C_VEL
LIN {X 0,Y 128.421,Z 563.39,A -85,B 0,C 180,E1 -25621.308,E2 -25621.308} C_VEL
LIN {X 0,Y 124.445,Z 568.862,A -85,B 0,C 180,E1 -25626.71,E2 -25626.71} C_VEL
LIN {X 0,Y 122.253,Z 572.373,A -85,B 0,C 180,E1 -25631.564,E2 -25631.564} C_VEL
LIN {X 0,Y 121.161,Z 574.931,A -85,B 0,C 180,E1 -25636.58,E2 -25636.58} C_VEL
LIN {X 0,Y 121.253,Z 576.915,A -85,B 0,C 180,E1 -25643.34,E2 -25643.34} C_VEL
LIN {X 0,Y 121.737,Z 577.292,A -85,B 0,C 180,E1 -25646.687,E2 -25646.687} C_VEL
LIN {X 0,Y 122.589,Z 577.231,A -85,B 0,C 180,E1 -25649.996,E2 -25649.996} C_VEL
LIN {X 0,Y 121.823,Z 576.49,A -85,B 0,C 180,E1 -25653.304,E2 -25653.304} C_VEL
LIN {X 0,Y 121.112,Z 574.049,A -85,B 0,C 180,E1 -25659.432,E2 -25659.432} C_VEL
LIN {X 0,Y 121.265,Z 570.45,A -85,B 0,C 180,E1 -25665.114,E2 -25665.114} C_VEL
LIN {X 0,Y 122.48,Z 566.116,A -85,B 0,C 180,E1 -25670.134,E2 -25670.134} C_VEL
LIN {X 0,Y 124.514,Z 560.862,A -85,B 0,C 180,E1 -25674.807,E2 -25674.807} C_VEL
LIN {X 0,Y 127.785,Z 553.721,A -85,B 0,C 180,E1 -25679.665,E2 -25679.665} C_VEL
LIN {X 0,Y 131.671,Z 545.232,A -85,B 0,C 180,E1 -25684.082,E2 -25684.082} C_VEL
LIN {X 0,Y 134.13,Z 535.779,A -85,B 0,C 180,E1 -25688.192,E2 -25688.192} C_VEL
LIN {X 0,Y 136.453,Z 526.31,A -85,B 0,C 180,E1 -25691.534,E2 -25691.534} C_VEL
LIN {X 0,Y 138.817,Z 515.851,A -85,B 0,C 180,E1 -25694.523,E2 -25694.523} C_VEL
LIN {X 0,Y 141.254,Z 503.879,A -85,B 0,C 180,E1 -25697.206,E2 -25697.206} C_VEL
LIN {X 0,Y 142.861,Z 493.351,A -85,B 0,C 180,E1 -25699.09,E2 -25699.09} C_VEL
LIN {X 0,Y 142.617,Z 480.759,A -85,B 0,C 180,E1 -25701.534,E2 -25701.534} C_VEL
LIN {X 0,Y 142.077,Z 475.494,A -85,B 0,C 180,E1 -25702.571,E2 -25702.571} C_VEL
LIN {X 0,Y 137.727,Z 464.887,A -85,B 0,C 180,E1 -25706.075,E2 -25706.075} C_VEL
LIN {X 0,Y 135.073,Z 459.093,A -85,B 0,C 180,E1 -25708.21,E2 -25708.21} C_VEL
LIN {X 0,Y 131.791,Z 452.821,A -85,B 0,C 180,E1 -25711.035,E2 -25711.035} C_VEL
LIN {X 0,Y 130.236,Z 449.835,A -85,B 0,C 180,E1 -25713.644,E2 -25713.644} C_VEL
LIN {X 0,Y 128.41,Z 448.075,A -85,B 0,C 180,E1 -25716.013,E2 -25716.013} C_VEL
LIN {X 0,Y 124.728,Z 446.589,A -85,B 0,C 180,E1 -25720.13,E2 -25720.13} C_VEL
LIN {X 0,Y 120.888,Z 445.177,A -85,B 0,C 180,E1 -25725.41,E2 -25725.41} C_VEL
LIN {X 0,Y 120.136,Z 444.329,A -85,B 0,C 180,E1 -25727.233,E2 -25727.233} C_VEL
LIN {X 0,Y 119.467,Z 442.895,A -85,B 0,C 180,E1 -25729.836,E2 -25729.836} C_VEL
LIN {X 0,Y 118.155,Z 438.914,A -85,B 0,C 180,E1 -25740.001,E2 -25740.001} C_VEL
LIN {X 0,Y 117.597,Z 439.026,A -85,B 0,C 180,E1 -25750.329,E2 -25750.329} C_VEL
LIN {X 0,Y 117.689,Z 439.604,A -85,B 0,C 180,E1 -25753.821,E2 -25753.821} C_VEL
LIN {X 0,Y 117.829,Z 440.691,A -85,B 0,C 180,E1 -25757.129,E2 -25757.129} C_VEL
LIN {X 0,Y 122.61,Z 445.268,A -85,B 0,C 180,E1 -25764.795,E2 -25764.795} C_VEL
LIN {X 0,Y 125.824,Z 449.119,A -85,B 0,C 180,E1 -25768.801,E2 -25768.801} C_VEL
LIN {X 0,Y 127.188,Z 450.892,A -85,B 0,C 180,E1 -25770.395,E2 -25770.395} C_VEL
LIN {X 0,Y 130.876,Z 456.184,A -85,B 0,C 180,E1 -25774.44,E2 -25774.44} C_VEL
LIN {X 0,Y 133.624,Z 460.865,A -85,B 0,C 180,E1 -25777.408,E2 -25777.408} C_VEL
LIN {X 0,Y 136.799,Z 467.172,A -85,B 0,C 180,E1 -25780.923,E2 -25780.923} C_VEL
LIN {X 0,Y 139.818,Z 474.824,A -85,B 0,C 180,E1 -25784.727,E2 -25784.727} C_VEL
LIN {X 0,Y 141.837,Z 482.021,A -85,B 0,C 180,E1 -25788.01,E2 -25788.01} C_VEL
LIN {X 0,Y 143.165,Z 489.424,A -85,B 0,C 180,E1 -25791.257,E2 -25791.257} C_VEL
LIN {X 0,Y 143.128,Z 490.568,A -85,B 0,C 180,E1 -25791.695,E2 -25791.695} C_VEL
LIN {X 0,Y 138.848,Z 501.107,A -85,B 0,C 180,E1 -25794.603,E2 -25794.603} C_VEL
LIN {X 0,Y 134.707,Z 509.767,A -85,B 0,C 180,E1 -25797.676,E2 -25797.676} C_VEL
LIN {X 0,Y 130.116,Z 518.505,A -85,B 0,C 180,E1 -25801.8,E2 -25801.8} C_VEL
LIN {X 0,Y 126.067,Z 525.55,A -85,B 0,C 180,E1 -25806.165,E2 -25806.165} C_VEL
LIN {X 0,Y 123.278,Z 530.295,A -85,B 0,C 180,E1 -25810.002,E2 -25810.002} C_VEL
LIN {X 0,Y 120.399,Z 534.909,A -85,B 0,C 180,E1 -25814.775,E2 -25814.775} C_VEL
LIN {X 0,Y 118.07,Z 538.454,A -85,B 0,C 180,E1 -25819.717,E2 -25819.717} C_VEL
LIN {X 0,Y 117.029,Z 540.271,A -85,B 0,C 180,E1 -25823.106,E2 -25823.106} C_VEL
LIN {X 0,Y 116.097,Z 542.584,A -85,B 0,C 180,E1 -25830.004,E2 -25830.004} C_VEL
LIN {X 0,Y 116.17,Z 543.166,A -85,B 0,C 180,E1 -25833.472,E2 -25833.472} C_VEL
LIN {X 0,Y 116.353,Z 543.393,A -85,B 0,C 180,E1 -25836.942,E2 -25836.942} C_VEL
LIN {X 0,Y 116.798,Z 543.211,A -85,B 0,C 180,E1 -25840.404,E2 -25840.404} C_VEL
LIN {X 0,Y 119.513,Z 541.603,A -85,B 0,C 180,E1 -25847.103,E2 -25847.103} C_VEL
LIN {X 0,Y 121.315,Z 540.191,A -85,B 0,C 180,E1 -25850.344,E2 -25850.344} C_VEL
LIN {X 0,Y 124.458,Z 537.122,A -85,B 0,C 180,E1 -25855.376,E2 -25855.376} C_VEL
LIN {X 0,Y 127.871,Z 533.432,A -85,B 0,C 180,E1 -25859.651,E2 -25859.651} C_VEL
LIN {X 0,Y 132.029,Z 528.382,A -85,B 0,C 180,E1 -25863.985,E2 -25863.985} C_VEL
LIN {X 0,Y 136.896,Z 521.981,A -85,B 0,C 180,E1 -25868.033,E2 -25868.033} C_VEL
LIN {X 0,Y 142.385,Z 513.672,A -85,B 0,C 180,E1 -25872.004,E2 -25872.004} C_VEL
LIN {X 0,Y 147.123,Z 505.727,A -85,B 0,C 180,E1 -25874.801,E2 -25874.801} C_VEL
LIN {X 0,Y 149.76,Z 500.56,A -85,B 0,C 180,E1 -25876.346,E2 -25876.346} C_VEL
LIN {X 0,Y 149.991,Z 499.133,A -85,B 0,C 180,E1 -25876.966,E2 -25876.966} C_VEL
LIN {X 0,Y 149.341,Z 492.158,A -85,B 0,C 180,E1 -25880.635,E2 -25880.635} C_VEL
LIN {X 0,Y 147.924,Z 485.362,A -85,B 0,C 180,E1 -25884.424,E2 -25884.424} C_VEL
LIN {X 0,Y 146.767,Z 481.511,A -85,B 0,C 180,E1 -25886.744,E2 -25886.744} C_VEL
LIN {X 0,Y 145.362,Z 481.064,A -85,B 0,C 180,E1 -25887.87,E2 -25887.87} C_VEL
LIN {X 0,Y 140.958,Z 483.462,A -85,B 0,C 180,E1 -25890.092,E2 -25890.092} C_VEL
LIN {X 0,Y 138.542,Z 485.24,A -85,B 0,C 180,E1 -25891.188,E2 -25891.188} C_VEL
LIN {X 0,Y 133.861,Z 489.202,A -85,B 0,C 180,E1 -25893.2,E2 -25893.2} C_VEL
LIN {X 0,Y 131.389,Z 490.863,A -85,B 0,C 180,E1 -25894.663,E2 -25894.663} C_VEL
LIN {X 0,Y 127.67,Z 493.062,A -85,B 0,C 180,E1 -25897.334,E2 -25897.334} C_VEL
LIN {X 0,Y 125.455,Z 494.95,A -85,B 0,C 180,E1 -25898.645,E2 -25898.645} C_VEL
LIN {X 0,Y 123.648,Z 496.26,A -85,B 0,C 180,E1 -25900.059,E2 -25900.059} C_VEL
LIN {X 0,Y 120.998,Z 497.67,A -85,B 0,C 180,E1 -25903.116,E2 -25903.116} C_VEL
LIN {X 0,Y 117.536,Z 500.876,A -85,B 0,C 180,E1 -25906.161,E2 -25906.161} C_VEL
LIN {X 0,Y 115.758,Z 502.032,A -85,B 0,C 180,E1 -25909.505,E2 -25909.505} C_VEL
LIN {X 0,Y 115.735,Z 502.056,A -85,B 0,C 180,E1 -25910.165,E2 -25910.165} C_VEL
LIN {X 0,Y 114.9,Z 512.912,A -85,B 0,C 180,E1 -25916.492,E2 -25916.492} C_VEL
LIN {X 0,Y 115.374,Z 521.88,A -85,B 0,C 180,E1 -25922.618,E2 -25922.618} C_VEL
LIN {X 0,Y 117.197,Z 531.479,A -85,B 0,C 180,E1 -25930.363,E2 -25930.363} C_VEL
LIN {X 0,Y 120.55,Z 538.664,A -85,B 0,C 180,E1 -25936.947,E2 -25936.947} C_VEL
LIN {X 0,Y 125.531,Z 544.724,A -85,B 0,C 180,E1 -25943.072,E2 -25943.072} C_VEL
LIN {X 0,Y 131.945,Z 549.736,A -85,B 0,C 180,E1 -25948.644,E2 -25948.644} C_VEL
LIN {X 0,Y 139.53,Z 553.761,A -85,B 0,C 180,E1 -25953.645,E2 -25953.645} C_VEL
LIN {X 0,Y 151.676,Z 557.844,A -85,B 0,C 180,E1 -25959.445,E2 -25959.445} C_VEL
LIN {X 0,Y 150.878,Z 558.405,A -85,B 0,C 180,E1 -25960.496,E2 -25960.496} C_VEL
LIN {X 0,Y 140.026,Z 560.084,A -85,B 0,C 180,E1 -25965.355,E2 -25965.355} C_VEL
LIN {X 0,Y 132.073,Z 560.989,A -85,B 0,C 180,E1 -25970.312,E2 -25970.312} C_VEL
LIN {X 0,Y 123.104,Z 561.393,A -85,B 0,C 180,E1 -25978.84,E2 -25978.84} C_VEL
LIN {X 0,Y 118.94,Z 566.516,A -85,B 0,C 180,E1 -25983.69,E2 -25983.69} C_VEL
LIN {X 0,Y 116.154,Z 570.344,A -85,B 0,C 180,E1 -25988.71,E2 -25988.71} C_VEL
LIN {X 0,Y 114.927,Z 572.367,A -85,B 0,C 180,E1 -25992.192,E2 -25992.192} C_VEL
LIN {X 0,Y 113.931,Z 575.109,A -85,B 0,C 180,E1 -25999.332,E2 -25999.332} C_VEL
LIN {X 0,Y 114.153,Z 575.905,A -85,B 0,C 180,E1 -26002.923,E2 -26002.923} C_VEL
LIN {X 0,Y 114.636,Z 576.273,A -85,B 0,C 180,E1 -26006.481,E2 -26006.481} C_VEL
LIN {X 0,Y 115.503,Z 576.206,A -85,B 0,C 180,E1 -26009.996,E2 -26009.996} C_VEL
LIN {X 0,Y 114.716,Z 575.453,A -85,B 0,C 180,E1 -26013.509,E2 -26013.509} C_VEL
LIN {X 0,Y 114.026,Z 573.198,A -85,B 0,C 180,E1 -26019.547,E2 -26019.547} C_VEL
LIN {X 0,Y 114.323,Z 569.357,A -85,B 0,C 180,E1 -26026.055,E2 -26026.055} C_VEL
LIN {X 0,Y 115.729,Z 565.002,A -85,B 0,C 180,E1 -26031.364,E2 -26031.364} C_VEL
LIN {X 0,Y 118.659,Z 558.405,A -85,B 0,C 180,E1 -26037.325,E2 -26037.325} C_VEL
LIN {X 0,Y 122.217,Z 551.296,A -85,B 0,C 180,E1 -26042.13,E2 -26042.13} C_VEL
LIN {X 0,Y 125.599,Z 544.015,A -85,B 0,C 180,E1 -26045.977,E2 -26045.977} C_VEL
LIN {X 0,Y 128.409,Z 533.91,A -85,B 0,C 180,E1 -26050.52,E2 -26050.52} C_VEL
LIN {X 0,Y 131.502,Z 522.72,A -85,B 0,C 180,E1 -26054.459,E2 -26054.459} C_VEL
LIN {X 0,Y 134.373,Z 511.115,A -85,B 0,C 180,E1 -26057.621,E2 -26057.621} C_VEL
LIN {X 0,Y 137.037,Z 498.381,A -85,B 0,C 180,E1 -26060.284,E2 -26060.284} C_VEL
LIN {X 0,Y 137.655,Z 493.218,A -85,B 0,C 180,E1 -26061.287,E2 -26061.287} C_VEL
LIN {X 0,Y 137.684,Z 481.249,A -85,B 0,C 180,E1 -26063.773,E2 -26063.773} C_VEL
LIN {X 0,Y 137.395,Z 479.025,A -85,B 0,C 180,E1 -26064.307,E2 -26064.307} C_VEL
LIN {X 0,Y 133.983,Z 469.538,A -85,B 0,C 180,E1 -26067.698,E2 -26067.698} C_VEL
LIN {X 0,Y 131.799,Z 464.238,A -85,B 0,C 180,E1 -26069.786,E2 -26069.786} C_VEL
LIN {X 0,Y 129.052,Z 458.603,A -85,B 0,C 180,E1 -26072.426,E2 -26072.426} C_VEL
LIN {X 0,Y 123.197,Z 450.486,A -85,B 0,C 180,E1 -26078.739,E2 -26078.739} C_VEL
LIN {X 0,Y 122.095,Z 448.041,A -85,B 0,C 180,E1 -26081.544,E2 -26081.544} C_VEL
LIN {X 0,Y 120.136,Z 444.329,A -85,B 0,C 180,E1 -26087.233,E2 -26087.233} C_VEL
LIN {X 0,Y 119.08,Z 443.33,A -85,B 0,C 180,E1 -26089.982,E2 -26089.982} C_VEL
LIN {X 0,Y 117.691,Z 443.131,A -85,B 0,C 180,E1 -26092.778,E2 -26092.778} C_VEL
LIN {X 0,Y 113.868,Z 444.368,A -85,B 0,C 180,E1 -26100.494,E2 -26100.494} C_VEL
LIN {X 0,Y 113.496,Z 444.622,A -85,B 0,C 180,E1 -26102.51,E2 -26102.51} C_VEL
LIN {X 0,Y 114.715,Z 445.692,A -85,B 0,C 180,E1 -26111.238,E2 -26111.238} C_VEL
LIN {X 0,Y 116.603,Z 447.572,A -85,B 0,C 180,E1 -26116.484,E2 -26116.484} C_VEL
LIN {X 0,Y 120.721,Z 451.906,A -85,B 0,C 180,E1 -26123.936,E2 -26123.936} C_VEL
LIN {X 0,Y 123.523,Z 455.617,A -85,B 0,C 180,E1 -26127.996,E2 -26127.996} C_VEL
LIN {X 0,Y 124.442,Z 456.953,A -85,B 0,C 180,E1 -26129.268,E2 -26129.268} C_VEL
LIN {X 0,Y 127.633,Z 462.036,A -85,B 0,C 180,E1 -26133.412,E2 -26133.412} C_VEL
LIN {X 0,Y 130.764,Z 468.086,A -85,B 0,C 180,E1 -26137.438,E2 -26137.438} C_VEL
LIN {X 0,Y 133.937,Z 476.125,A -85,B 0,C 180,E1 -26141.993,E2 -26141.993} C_VEL
LIN {X 0,Y 135.824,Z 482.71,A -85,B 0,C 180,E1 -26145.355,E2 -26145.355} C_VEL
LIN {X 0,Y 137.1,Z 489.441,A -85,B 0,C 180,E1 -26148.597,E2 -26148.597} C_VEL
LIN {X 0,Y 137.381,Z 491.91,A -85,B 0,C 180,E1 -26149.776,E2 -26149.776} C_VEL
LIN {X 0,Y 137.22,Z 493.078,A -85,B 0,C 180,E1 -26150.199,E2 -26150.199} C_VEL
LIN {X 0,Y 133.281,Z 502.159,A -85,B 0,C 180,E1 -26152.806,E2 -26152.806} C_VEL
LIN {X 0,Y 128.837,Z 510.941,A -85,B 0,C 180,E1 -26156.009,E2 -26156.009} C_VEL
LIN {X 0,Y 123.983,Z 519.649,A -85,B 0,C 180,E1 -26160.269,E2 -26160.269} C_VEL
LIN {X 0,Y 119.691,Z 526.67,A -85,B 0,C 180,E1 -26164.809,E2 -26164.809} C_VEL
LIN {X 0,Y 116.713,Z 531.393,A -85,B 0,C 180,E1 -26168.824,E2 -26168.824} C_VEL
LIN {X 0,Y 113.656,Z 535.985,A -85,B 0,C 180,E1 -26173.848,E2 -26173.848} C_VEL
LIN {X 0,Y 111.166,Z 539.514,A -85,B 0,C 180,E1 -26179.071,E2 -26179.071} C_VEL
LIN {X 0,Y 110.058,Z 541.319,A -85,B 0,C 180,E1 -26182.667,E2 -26182.667} C_VEL
LIN {X 0,Y 109.069,Z 543.609,A -85,B 0,C 180,E1 -26190.004,E2 -26190.004} C_VEL
LIN {X 0,Y 109.155,Z 544.184,A -85,B 0,C 180,E1 -26193.696,E2 -26193.696} C_VEL
LIN {X 0,Y 109.376,Z 544.395,A -85,B 0,C 180,E1 -26197.387,E2 -26197.387} C_VEL
LIN {X 0,Y 109.887,Z 544.203,A -85,B 0,C 180,E1 -26201.066,E2 -26201.066} C_VEL
LIN {X 0,Y 112.813,Z 542.577,A -85,B 0,C 180,E1 -26208.153,E2 -26208.153} C_VEL
LIN {X 0,Y 114.747,Z 541.147,A -85,B 0,C 180,E1 -26211.564,E2 -26211.564} C_VEL
LIN {X 0,Y 118.137,Z 538.066,A -85,B 0,C 180,E1 -26216.827,E2 -26216.827} C_VEL
LIN {X 0,Y 121.795,Z 534.349,A -85,B 0,C 180,E1 -26221.291,E2 -26221.291} C_VEL
LIN {X 0,Y 126.254,Z 529.276,A -85,B 0,C 180,E1 -26225.771,E2 -26225.771} C_VEL
LIN {X 0,Y 131.418,Z 522.85,A -85,B 0,C 180,E1 -26229.926,E2 -26229.926} C_VEL
LIN {X 0,Y 137.188,Z 514.571,A -85,B 0,C 180,E1 -26233.944,E2 -26233.944} C_VEL
LIN {X 0,Y 142.208,Z 506.514,A -85,B 0,C 180,E1 -26236.803,E2 -26236.803} C_VEL
LIN {X 0,Y 143.957,Z 503.369,A -85,B 0,C 180,E1 -26237.771,E2 -26237.771} C_VEL
LIN {X 0,Y 144.354,Z 502.067,A -85,B 0,C 180,E1 -26238.289,E2 -26238.289} C_VEL
LIN {X 0,Y 143.94,Z 494.859,A -85,B 0,C 180,E1 -26242.422,E2 -26242.422} C_VEL
LIN {X 0,Y 142.786,Z 488.493,A -85,B 0,C 180,E1 -26246.339,E2 -26246.339} C_VEL
LIN {X 0,Y 142.409,Z 487.615,A -85,B 0,C 180,E1 -26247.035,E2 -26247.035} C_VEL
LIN {X 0,Y 139.986,Z 488.838,A -85,B 0,C 180,E1 -26248.186,E2 -26248.186} C_VEL
LIN {X 0,Y 137.428,Z 490.547,A -85,B 0,C 180,E1 -26249.242,E2 -26249.242} C_VEL
LIN {X 0,Y 132.089,Z 494.623,A -85,B 0,C 180,E1 -26251.388,E2 -26251.388} C_VEL
LIN {X 0,Y 125.807,Z 498.204,A -85,B 0,C 180,E1 -26255.229,E2 -26255.229} C_VEL
LIN {X 0,Y 123.498,Z 499.947,A -85,B 0,C 180,E1 -26256.524,E2 -26256.524} C_VEL
LIN {X 0,Y 121.115,Z 501.563,A -85,B 0,C 180,E1 -26258.2,E2 -26258.2} C_VEL
LIN {X 0,Y 118.416,Z 502.947,A -85,B 0,C 180,E1 -26260.947,E2 -26260.947} C_VEL
LIN {X 0,Y 114.785,Z 505.785,A -85,B 0,C 180,E1 -26264.006,E2 -26264.006} C_VEL
LIN {X 0,Y 113.462,Z 506.708,A -85,B 0,C 180,E1 -26265.654,E2 -26265.654} C_VEL
LIN {X 0,Y 111.485,Z 508.047,A -85,B 0,C 180,E1 -26269.098,E2 -26269.098} C_VEL
LIN {X 0,Y 109.961,Z 509.637,A -85,B 0,C 180,E1 -26270.805,E2 -26270.805} C_VEL
LIN {X 0,Y 108.805,Z 510.853,A -85,B 0,C 180,E1 -26272.577,E2 -26272.577} C_VEL
LIN {X 0,Y 107.886,Z 511.936,A -85,B 0,C 180,E1 -26276.731,E2 -26276.731} C_VEL
LIN {X 0,Y 107.918,Z 512.333,A -85,B 0,C 180,E1 -26277.199,E2 -26277.199} C_VEL
LIN {X 0,Y 108.518,Z 521.471,A -85,B 0,C 180,E1 -26283.712,E2 -26283.712} C_VEL
LIN {X 0,Y 110.673,Z 531.351,A -85,B 0,C 180,E1 -26291.91,E2 -26291.91} C_VEL
LIN {X 0,Y 115.006,Z 539.578,A -85,B 0,C 180,E1 -26299.639,E2 -26299.639} C_VEL
LIN {X 0,Y 122.19,Z 547.042,A -85,B 0,C 180,E1 -26307.395,E2 -26307.395} C_VEL
LIN {X 0,Y 131.606,Z 552.971,A -85,B 0,C 180,E1 -26314.105,E2 -26314.105} C_VEL
LIN {X 0,Y 142.786,Z 557.504,A -85,B 0,C 180,E1 -26319.781,E2 -26319.781} C_VEL
LIN {X 0,Y 130.851,Z 558.796,A -85,B 0,C 180,E1 -26325.711,E2 -26325.711} C_VEL
LIN {X 0,Y 119.962,Z 559.054,A -85,B 0,C 180,E1 -26334.133,E2 -26334.133} C_VEL
LIN {X 0,Y 118.323,Z 559.084,A -85,B 0,C 180,E1 -26335.902,E2 -26335.902} C_VEL
LIN {X 0,Y 113.919,Z 564.092,A -85,B 0,C 180,E1 -26340.422,E2 -26340.422} C_VEL
LIN {X 0,Y 110.433,Z 568.237,A -85,B 0,C 180,E1 -26345.561,E2 -26345.561} C_VEL
LIN {X 0,Y 108.138,Z 571.386,A -85,B 0,C 180,E1 -26351.033,E2 -26351.033} C_VEL
LIN {X 0,Y 106.895,Z 574.106,A -85,B 0,C 180,E1 -26358.62,E2 -26358.62} C_VEL
LIN {X 0,Y 107.044,Z 574.894,A -85,B 0,C 180,E1 -26362.451,E2 -26362.451} C_VEL
LIN {X 0,Y 107.535,Z 575.252,A -85,B 0,C 180,E1 -26366.249,E2 -26366.249} C_VEL
LIN {X 0,Y 108.418,Z 575.182,A -85,B 0,C 180,E1 -26369.996,E2 -26369.996} C_VEL
LIN {X 0,Y 107.608,Z 574.414,A -85,B 0,C 180,E1 -26373.741,E2 -26373.741} C_VEL
LIN {X 0,Y 106.958,Z 572.325,A -85,B 0,C 180,E1 -26379.732,E2 -26379.732} C_VEL
LIN {X 0,Y 107.113,Z 569.467,A -85,B 0,C 180,E1 -26385.211,E2 -26385.211} C_VEL
LIN {X 0,Y 108.376,Z 565.462,A -85,B 0,C 180,E1 -26390.891,E2 -26390.891} C_VEL
LIN {X 0,Y 110.733,Z 560.32,A -85,B 0,C 180,E1 -26396.372,E2 -26396.372} C_VEL
LIN {X 0,Y 114.151,Z 553.903,A -85,B 0,C 180,E1 -26401.551,E2 -26401.551} C_VEL
LIN {X 0,Y 118.407,Z 545.913,A -85,B 0,C 180,E1 -26406.404,E2 -26406.404} C_VEL
LIN {X 0,Y 121.365,Z 537.064,A -85,B 0,C 180,E1 -26410.892,E2 -26410.892} C_VEL
LIN {X 0,Y 124.108,Z 528.328,A -85,B 0,C 180,E1 -26414.484,E2 -26414.484} C_VEL
LIN {X 0,Y 127.63,Z 516.488,A -85,B 0,C 180,E1 -26418.319,E2 -26418.319} C_VEL
LIN {X 0,Y 130.68,Z 504.637,A -85,B 0,C 180,E1 -26421.237,E2 -26421.237} C_VEL
LIN {X 0,Y 132.498,Z 495.56,A -85,B 0,C 180,E1 -26423.094,E2 -26423.094} C_VEL
LIN {X 0,Y 132.944,Z 483.636,A -85,B 0,C 180,E1 -26425.769,E2 -26425.769} C_VEL
LIN {X 0,Y 130.853,Z 476.194,A -85,B 0,C 180,E1 -26428.513,E2 -26428.513} C_VEL
LIN {X 0,Y 128.431,Z 469.33,A -85,B 0,C 180,E1 -26431.393,E2 -26431.393} C_VEL
LIN {X 0,Y 126.264,Z 464.302,A -85,B 0,C 180,E1 -26433.892,E2 -26433.892} C_VEL
LIN {X 0,Y 120.823,Z 456.298,A -85,B 0,C 180,E1 -26440.461,E2 -26440.461} C_VEL
LIN {X 0,Y 118.228,Z 452.855,A -85,B 0,C 180,E1 -26444.485,E2 -26444.485} C_VEL
LIN {X 0,Y 115.536,Z 448.724,A -85,B 0,C 180,E1 -26450.371,E2 -26450.371} C_VEL
LIN {X 0,Y 113.796,Z 445.203,A -85,B 0,C 180,E1 -26458.231,E2 -26458.231} C_VEL
LIN {X 0,Y 113.8,Z 444.597,A -85,B 0,C 180,E1 -26460.001,E2 -26460.001} C_VEL
LIN {X 0,Y 113.496,Z 444.622,A -85,B 0,C 180,E1 -26462.51,E2 -26462.51} C_VEL
LIN {X 0,Y 113.555,Z 445.506,A -85,B 0,C 180,E1 -26465.463,E2 -26465.463} C_VEL
LIN {X 0,Y 113.77,Z 447.345,A -85,B 0,C 180,E1 -26468.313,E2 -26468.313} C_VEL
LIN {X 0,Y 115.745,Z 455.366,A -85,B 0,C 180,E1 -26477.472,E2 -26477.472} C_VEL
LIN {X 0,Y 118.563,Z 458.519,A -85,B 0,C 180,E1 -26483.124,E2 -26483.124} C_VEL
LIN {X 0,Y 121.108,Z 462.17,A -85,B 0,C 180,E1 -26487.428,E2 -26487.428} C_VEL
LIN {X 0,Y 124.187,Z 467.772,A -85,B 0,C 180,E1 -26492.331,E2 -26492.331} C_VEL
LIN {X 0,Y 126.959,Z 473.96,A -85,B 0,C 180,E1 -26496.715,E2 -26496.715} C_VEL
LIN {X 0,Y 129.497,Z 481.658,A -85,B 0,C 180,E1 -26501.377,E2 -26501.377} C_VEL
LIN {X 0,Y 131.067,Z 488.767,A -85,B 0,C 180,E1 -26505.276,E2 -26505.276} C_VEL
LIN {X 0,Y 131.742,Z 494.684,A -85,B 0,C 180,E1 -26508.32,E2 -26508.32} C_VEL
LIN {X 0,Y 126.9,Z 505.093,A -85,B 0,C 180,E1 -26511.5,E2 -26511.5} C_VEL
LIN {X 0,Y 122.188,Z 513.683,A -85,B 0,C 180,E1 -26514.893,E2 -26514.893} C_VEL
LIN {X 0,Y 117.17,Z 522.09,A -85,B 0,C 180,E1 -26519.351,E2 -26519.351} C_VEL
LIN {X 0,Y 112.688,Z 528.798,A -85,B 0,C 180,E1 -26524.12,E2 -26524.12} C_VEL
LIN {X 0,Y 109.027,Z 534.141,A -85,B 0,C 180,E1 -26529.24,E2 -26529.24} C_VEL
LIN {X 0,Y 106.004,Z 538.335,A -85,B 0,C 180,E1 -26534.626,E2 -26534.626} C_VEL
LIN {X 0,Y 104.278,Z 540.575,A -85,B 0,C 180,E1 -26538.339,E2 -26538.339} C_VEL
LIN {X 0,Y 103.095,Z 542.365,A -85,B 0,C 180,E1 -26542.168,E2 -26542.168} C_VEL
LIN {X 0,Y 102.041,Z 544.635,A -85,B 0,C 180,E1 -26550.004,E2 -26550.004} C_VEL
LIN {X 0,Y 102.141,Z 545.201,A -85,B 0,C 180,E1 -26553.95,E2 -26553.95} C_VEL
LIN {X 0,Y 102.407,Z 545.395,A -85,B 0,C 180,E1 -26557.893,E2 -26557.893} C_VEL
LIN {X 0,Y 102.992,Z 545.195,A -85,B 0,C 180,E1 -26561.817,E2 -26561.817} C_VEL
LIN {X 0,Y 106.155,Z 543.549,A -85,B 0,C 180,E1 -26569.335,E2 -26569.335} C_VEL
LIN {X 0,Y 108.238,Z 542.103,A -85,B 0,C 180,E1 -26572.933,E2 -26572.933} C_VEL
LIN {X 0,Y 111.831,Z 539.061,A -85,B 0,C 180,E1 -26578.376,E2 -26578.376} C_VEL
LIN {X 0,Y 115.832,Z 535.267,A -85,B 0,C 180,E1 -26583.102,E2 -26583.102} C_VEL
LIN {X 0,Y 120.615,Z 530.169,A -85,B 0,C 180,E1 -26587.725,E2 -26587.725} C_VEL
LIN {X 0,Y 126.096,Z 523.72,A -85,B 0,C 180,E1 -26591.981,E2 -26591.981} C_VEL
LIN {X 0,Y 132.101,Z 515.542,A -85,B 0,C 180,E1 -26596.009,E2 -26596.009} C_VEL
LIN {X 0,Y 137.476,Z 507.302,A -85,B 0,C 180,E1 -26598.946,E2 -26598.946} C_VEL
LIN {X 0,Y 138.595,Z 505.41,A -85,B 0,C 180,E1 -26599.524,E2 -26599.524} C_VEL
LIN {X 0,Y 138.808,Z 501.584,A -85,B 0,C 180,E1 -26601.804,E2 -26601.804} C_VEL
LIN {X 0,Y 138.499,Z 496.371,A -85,B 0,C 180,E1 -26605.132,E2 -26605.132} C_VEL
LIN {X 0,Y 138.313,Z 495.037,A -85,B 0,C 180,E1 -26606.017,E2 -26606.017} C_VEL
LIN {X 0,Y 136.228,Z 495.657,A -85,B 0,C 180,E1 -26607.2,E2 -26607.2} C_VEL
LIN {X 0,Y 131.097,Z 499.217,A -85,B 0,C 180,E1 -26609.07,E2 -26609.07} C_VEL
LIN {X 0,Y 128.182,Z 500.924,A -85,B 0,C 180,E1 -26610.431,E2 -26610.431} C_VEL
LIN {X 0,Y 123.86,Z 503.147,A -85,B 0,C 180,E1 -26613.003,E2 -26613.003} C_VEL
LIN {X 0,Y 119.268,Z 506.108,A -85,B 0,C 180,E1 -26615.638,E2 -26615.638} C_VEL
LIN {X 0,Y 113.896,Z 509.079,A -85,B 0,C 180,E1 -26620.16,E2 -26620.16} C_VEL
LIN {X 0,Y 111.952,Z 510.474,A -85,B 0,C 180,E1 -26621.705,E2 -26621.705} C_VEL
LIN {X 0,Y 106.543,Z 514.221,A -85,B 0,C 180,E1 -26628.585,E2 -26628.585} C_VEL
LIN {X 0,Y 105.143,Z 515.465,A -85,B 0,C 180,E1 -26630.379,E2 -26630.379} C_VEL
LIN {X 0,Y 104.205,Z 516.312,A -85,B 0,C 180,E1 -26632.247,E2 -26632.247} C_VEL
LIN {X 0,Y 103.167,Z 517.461,A -85,B 0,C 180,E1 -26636.093,E2 -26636.093} C_VEL
LIN {X 0,Y 101.611,Z 519.706,A -85,B 0,C 180,E1 -26639.999,E2 -26639.999} C_VEL
LIN {X 0,Y 101.457,Z 520.943,A -85,B 0,C 180,E1 -26643.971,E2 -26643.971} C_VEL
LIN {X 0,Y 101.725,Z 521.264,A -85,B 0,C 180,E1 -26645.202,E2 -26645.202} C_VEL
LIN {X 0,Y 104.239,Z 531.051,A -85,B 0,C 180,E1 -26653.648,E2 -26653.648} C_VEL
LIN {X 0,Y 108.392,Z 538.632,A -85,B 0,C 180,E1 -26660.891,E2 -26660.891} C_VEL
LIN {X 0,Y 115.946,Z 546.549,A -85,B 0,C 180,E1 -26669.006,E2 -26669.006} C_VEL
LIN {X 0,Y 125.796,Z 552.94,A -85,B 0,C 180,E1 -26675.916,E2 -26675.916} C_VEL
LIN {X 0,Y 132.591,Z 556.096,A -85,B 0,C 180,E1 -26679.498,E2 -26679.498} C_VEL
LIN {X 0,Y 130.524,Z 556.536,A -85,B 0,C 180,E1 -26681.073,E2 -26681.073} C_VEL
LIN {X 0,Y 117.959,Z 556.861,A -85,B 0,C 180,E1 -26689.047,E2 -26689.047} C_VEL
LIN {X 0,Y 113.932,Z 556.664,A -85,B 0,C 180,E1 -26692.746,E2 -26692.746} C_VEL
LIN {X 0,Y 108.93,Z 561.908,A -85,B 0,C 180,E1 -26697.26,E2 -26697.26} C_VEL
LIN {X 0,Y 105.07,Z 565.988,A -85,B 0,C 180,E1 -26702.077,E2 -26702.077} C_VEL
LIN {X 0,Y 102.967,Z 568.411,A -85,B 0,C 180,E1 -26705.82,E2 -26705.82} C_VEL
LIN {X 0,Y 101.388,Z 570.401,A -85,B 0,C 180,E1 -26709.717,E2 -26709.717} C_VEL
LIN {X 0,Y 99.89,Z 573.104,A -85,B 0,C 180,E1 -26717.811,E2 -26717.811} C_VEL
LIN {X 0,Y 99.948,Z 573.882,A -85,B 0,C 180,E1 -26721.911,E2 -26721.911} C_VEL
LIN {X 0,Y 100.433,Z 574.231,A -85,B 0,C 180,E1 -26725.983,E2 -26725.983} C_VEL
LIN {X 0,Y 101.301,Z 574.152,A -85,B 0,C 180,E1 -26729.996,E2 -26729.996} C_VEL
LIN {X 0,Y 100.498,Z 573.376,A -85,B 0,C 180,E1 -26734.006,E2 -26734.006} C_VEL
LIN {X 0,Y 99.88,Z 571.465,A -85,B 0,C 180,E1 -26739.907,E2 -26739.907} C_VEL
LIN {X 0,Y 100.191,Z 568.386,A -85,B 0,C 180,E1 -26746.29,E2 -26746.29} C_VEL
LIN {X 0,Y 101.672,Z 564.359,A -85,B 0,C 180,E1 -26752.34,E2 -26752.34} C_VEL
LIN {X 0,Y 104.311,Z 559.196,A -85,B 0,C 180,E1 -26758.135,E2 -26758.135} C_VEL
LIN {X 0,Y 108.074,Z 552.761,A -85,B 0,C 180,E1 -26763.551,E2 -26763.551} C_VEL
LIN {X 0,Y 111.859,Z 546.201,A -85,B 0,C 180,E1 -26767.771,E2 -26767.771} C_VEL
LIN {X 0,Y 114.942,Z 538.071,A -85,B 0,C 180,E1 -26772.261,E2 -26772.261} C_VEL
LIN {X 0,Y 118.073,Z 529.253,A -85,B 0,C 180,E1 -26776.19,E2 -26776.19} C_VEL
LIN {X 0,Y 121.782,Z 518.178,A -85,B 0,C 180,E1 -26780.035,E2 -26780.035} C_VEL
LIN {X 0,Y 125.122,Z 507.017,A -85,B 0,C 180,E1 -26783.029,E2 -26783.029} C_VEL
LIN {X 0,Y 127.309,Z 498.327,A -85,B 0,C 180,E1 -26784.9,E2 -26784.9} C_VEL
LIN {X 0,Y 128.275,Z 486.727,A -85,B 0,C 180,E1 -26787.712,E2 -26787.712} C_VEL
LIN {X 0,Y 126.485,Z 479.52,A -85,B 0,C 180,E1 -26790.68,E2 -26790.68} C_VEL
LIN {X 0,Y 124.798,Z 473.953,A -85,B 0,C 180,E1 -26793.224,E2 -26793.224} C_VEL
LIN {X 0,Y 123.313,Z 469.914,A -85,B 0,C 180,E1 -26795.37,E2 -26795.37} C_VEL
LIN {X 0,Y 118.686,Z 462.396,A -85,B 0,C 180,E1 -26801.889,E2 -26801.889} C_VEL
LIN {X 0,Y 115.262,Z 457.163,A -85,B 0,C 180,E1 -26808.543,E2 -26808.543} C_VEL
LIN {X 0,Y 113.573,Z 454.346,A -85,B 0,C 180,E1 -26813.784,E2 -26813.784} C_VEL
LIN {X 0,Y 112.714,Z 451.719,A -85,B 0,C 180,E1 -26820.001,E2 -26820.001} C_VEL
LIN {X 0,Y 113.035,Z 452.169,A -85,B 0,C 180,E1 -26828.043,E2 -26828.043} C_VEL
LIN {X 0,Y 114.41,Z 453.485,A -85,B 0,C 180,E1 -26833.646,E2 -26833.646} C_VEL
LIN {X 0,Y 115.569,Z 455.109,A -85,B 0,C 180,E1 -26837.018,E2 -26837.018} C_VEL
LIN {X 0,Y 115.745,Z 455.366,A -85,B 0,C 180,E1 -26837.472,E2 -26837.472} C_VEL
LIN {X 0,Y 116.719,Z 457.78,A -85,B 0,C 180,E1 -26840.096,E2 -26840.096} C_VEL
LIN {X 0,Y 117.955,Z 463.276,A -85,B 0,C 180,E1 -26844.088,E2 -26844.088} C_VEL
LIN {X 0,Y 118.876,Z 468.086,A -85,B 0,C 180,E1 -26847.171,E2 -26847.171} C_VEL
LIN {X 0,Y 120.153,Z 472.38,A -85,B 0,C 180,E1 -26850.358,E2 -26850.358} C_VEL
LIN {X 0,Y 122.487,Z 478.3,A -85,B 0,C 180,E1 -26855.015,E2 -26855.015} C_VEL
LIN {X 0,Y 124.413,Z 485.03,A -85,B 0,C 180,E1 -26859.495,E2 -26859.495} C_VEL
LIN {X 0,Y 125.62,Z 491.427,A -85,B 0,C 180,E1 -26863.345,E2 -26863.345} C_VEL
LIN {X 0,Y 126.078,Z 496.914,A -85,B 0,C 180,E1 -26866.442,E2 -26866.442} C_VEL
LIN {X 0,Y 121.527,Z 506.244,A -85,B 0,C 180,E1 -26869.425,E2 -26869.425} C_VEL
LIN {X 0,Y 116.525,Z 514.855,A -85,B 0,C 180,E1 -26872.911,E2 -26872.911} C_VEL
LIN {X 0,Y 111.195,Z 523.227,A -85,B 0,C 180,E1 -26877.509,E2 -26877.509} C_VEL
LIN {X 0,Y 106.427,Z 529.907,A -85,B 0,C 180,E1 -26882.473,E2 -26882.473} C_VEL
LIN {X 0,Y 102.495,Z 535.23,A -85,B 0,C 180,E1 -26887.849,E2 -26887.849} C_VEL
LIN {X 0,Y 99.263,Z 539.403,A -85,B 0,C 180,E1 -26893.553,E2 -26893.553} C_VEL
LIN {X 0,Y 97.409,Z 541.636,A -85,B 0,C 180,E1 -26897.504,E2 -26897.504} C_VEL
LIN {X 0,Y 96.14,Z 543.409,A -85,B 0,C 180,E1 -26901.598,E2 -26901.598} C_VEL
LIN {X 0,Y 95.013,Z 545.661,A -85,B 0,C 180,E1 -26910.005,E2 -26910.005} C_VEL
LIN {X 0,Y 95.129,Z 546.219,A -85,B 0,C 180,E1 -26914.241,E2 -26914.241} C_VEL
LIN {X 0,Y 95.447,Z 546.395,A -85,B 0,C 180,E1 -26918.473,E2 -26918.473} C_VEL
LIN {X 0,Y 96.118,Z 546.187,A -85,B 0,C 180,E1 -26922.676,E2 -26922.676} C_VEL
LIN {X 0,Y 99.549,Z 544.52,A -85,B 0,C 180,E1 -26930.675,E2 -26930.675} C_VEL
LIN {X 0,Y 101.799,Z 543.058,A -85,B 0,C 180,E1 -26934.475,E2 -26934.475} C_VEL
LIN {X 0,Y 105.571,Z 540.087,A -85,B 0,C 180,E1 -26940.067,E2 -26940.067} C_VEL
LIN {X 0,Y 109.996,Z 536.185,A -85,B 0,C 180,E1 -26945.107,E2 -26945.107} C_VEL
LIN {X 0,Y 115.131,Z 531.063,A -85,B 0,C 180,E1 -26949.868,E2 -26949.868} C_VEL
LIN {X 0,Y 120.95,Z 524.589,A -85,B 0,C 180,E1 -26954.214,E2 -26954.214} C_VEL
LIN {X 0,Y 127.212,Z 516.499,A -85,B 0,C 180,E1 -26958.242,E2 -26958.242} C_VEL
LIN {X 0,Y 132.961,Z 508.089,A -85,B 0,C 180,E1 -26961.233,E2 -26961.233} C_VEL
LIN {X 0,Y 133.437,Z 505.005,A -85,B 0,C 180,E1 -26963.141,E2 -26963.141} C_VEL
LIN {X 0,Y 133.452,Z 501.574,A -85,B 0,C 180,E1 -26965.518,E2 -26965.518} C_VEL
LIN {X 0,Y 126.961,Z 505.376,A -85,B 0,C 180,E1 -26967.945,E2 -26967.945} C_VEL
LIN {X 0,Y 121.852,Z 507.889,A -85,B 0,C 180,E1 -26970.644,E2 -26970.644} C_VEL
LIN {X 0,Y 116.981,Z 510.675,A -85,B 0,C 180,E1 -26973.218,E2 -26973.218} C_VEL
LIN {X 0,Y 111.131,Z 513.63,A -85,B 0,C 180,E1 -26977.7,E2 -26977.7} C_VEL
LIN {X 0,Y 107.308,Z 515.985,A -85,B 0,C 180,E1 -26980.884,E2 -26980.884} C_VEL
LIN {X 0,Y 102.895,Z 518.699,A -85,B 0,C 180,E1 -26986.168,E2 -26986.168} C_VEL
LIN {X 0,Y 99.606,Z 521.271,A -85,B 0,C 180,E1 -26991.071,E2 -26991.071} C_VEL
LIN {X 0,Y 97.887,Z 523.009,A -85,B 0,C 180,E1 -26995.882,E2 -26995.882} C_VEL
LIN {X 0,Y 96.607,Z 524.854,A -85,B 0,C 180,E1 -26999.999,E2 -26999.999} C_VEL
LIN {X 0,Y 96.513,Z 526.014,A -85,B 0,C 180,E1 -27004.175,E2 -27004.175} C_VEL
LIN {X 0,Y 95.928,Z 528.112,A -85,B 0,C 180,E1 -27008.425,E2 -27008.425} C_VEL
LIN {X 0,Y 96.529,Z 529.58,A -85,B 0,C 180,E1 -27012.615,E2 -27012.615} C_VEL
LIN {X 0,Y 97.713,Z 530.115,A -85,B 0,C 180,E1 -27015.112,E2 -27015.112} C_VEL
LIN {X 0,Y 103.224,Z 539.327,A -85,B 0,C 180,E1 -27024.11,E2 -27024.11} C_VEL
LIN {X 0,Y 111.793,Z 547.35,A -85,B 0,C 180,E1 -27032.3,E2 -27032.3} C_VEL
LIN {X 0,Y 123.177,Z 554.261,A -85,B 0,C 180,E1 -27039.594,E2 -27039.594} C_VEL
LIN {X 0,Y 122.571,Z 554.589,A -85,B 0,C 180,E1 -27040.563,E2 -27040.563} C_VEL
LIN {X 0,Y 111.061,Z 554.328,A -85,B 0,C 180,E1 -27048.356,E2 -27048.356} C_VEL
LIN {X 0,Y 109.942,Z 554.227,A -85,B 0,C 180,E1 -27049.361,E2 -27049.361} C_VEL
LIN {X 0,Y 103.744,Z 560.262,A -85,B 0,C 180,E1 -27054.381,E2 -27054.381} C_VEL
LIN {X 0,Y 98.817,Z 565.032,A -85,B 0,C 180,E1 -27060.138,E2 -27060.138} C_VEL
LIN {X 0,Y 96.494,Z 567.446,A -85,B 0,C 180,E1 -27064.083,E2 -27064.083} C_VEL
LIN {X 0,Y 94.714,Z 569.417,A -85,B 0,C 180,E1 -27068.217,E2 -27068.217} C_VEL
LIN {X 0,Y 92.911,Z 572.102,A -85,B 0,C 180,E1 -27076.879,E2 -27076.879} C_VEL
LIN {X 0,Y 92.859,Z 572.871,A -85,B 0,C 180,E1 -27081.289,E2 -27081.289} C_VEL
LIN {X 0,Y 93.331,Z 573.209,A -85,B 0,C 180,E1 -27085.677,E2 -27085.677} C_VEL
LIN {X 0,Y 94.182,Z 573.123,A -85,B 0,C 180,E1 -27089.995,E2 -27089.995} C_VEL
LIN {X 0,Y 93.353,Z 572.331,A -85,B 0,C 180,E1 -27094.313,E2 -27094.313} C_VEL
LIN {X 0,Y 92.808,Z 570.6,A -85,B 0,C 180,E1 -27100.126,E2 -27100.126} C_VEL
LIN {X 0,Y 93.287,Z 567.3,A -85,B 0,C 180,E1 -27107.534,E2 -27107.534} C_VEL
LIN {X 0,Y 95.053,Z 563.258,A -85,B 0,C 180,E1 -27113.99,E2 -27113.99} C_VEL
LIN {X 0,Y 98.022,Z 558.074,A -85,B 0,C 180,E1 -27120.119,E2 -27120.119} C_VEL
LIN {X 0,Y 102.138,Z 551.615,A -85,B 0,C 180,E1 -27125.788,E2 -27125.788} C_VEL
LIN {X 0,Y 106.082,Z 544.997,A -85,B 0,C 180,E1 -27130.231,E2 -27130.231} C_VEL
LIN {X 0,Y 109.574,Z 536.434,A -85,B 0,C 180,E1 -27135.129,E2 -27135.129} C_VEL
LIN {X 0,Y 113.831,Z 525.721,A -85,B 0,C 180,E1 -27139.815,E2 -27139.815} C_VEL
LIN {X 0,Y 118.022,Z 514.22,A -85,B 0,C 180,E1 -27143.641,E2 -27143.641} C_VEL
LIN {X 0,Y 121.739,Z 502.296,A -85,B 0,C 180,E1 -27146.611,E2 -27146.611} C_VEL
LIN {X 0,Y 122.724,Z 497.671,A -85,B 0,C 180,E1 -27147.731,E2 -27147.731} C_VEL
LIN {X 0,Y 123.635,Z 490.037,A -85,B 0,C 180,E1 -27149.703,E2 -27149.703} C_VEL
LIN {X 0,Y 122.732,Z 485.24,A -85,B 0,C 180,E1 -27151.809,E2 -27151.809} C_VEL
LIN {X 0,Y 121.142,Z 478.695,A -85,B 0,C 180,E1 -27155.014,E2 -27155.014} C_VEL
LIN {X 0,Y 120.082,Z 475.349,A -85,B 0,C 180,E1 -27156.966,E2 -27156.966} C_VEL
LIN {X 0,Y 116.345,Z 468.531,A -85,B 0,C 180,E1 -27163.242,E2 -27163.242} C_VEL
LIN {X 0,Y 113.192,Z 463.066,A -85,B 0,C 180,E1 -27170.705,E2 -27170.705} C_VEL
LIN {X 0,Y 111.597,Z 458.939,A -85,B 0,C 180,E1 -27179.697,E2 -27179.697} C_VEL
LIN {X 0,Y 111.503,Z 458.894,A -85,B 0,C 180,E1 -27185.426,E2 -27185.426} C_VEL
LIN {X 0,Y 112.477,Z 459.866,A -85,B 0,C 180,E1 -27191.718,E2 -27191.718} C_VEL
LIN {X 0,Y 113.504,Z 461.484,A -85,B 0,C 180,E1 -27195.718,E2 -27195.718} C_VEL
LIN {X 0,Y 116.19,Z 465.122,A -85,B 0,C 180,E1 -27202.448,E2 -27202.448} C_VEL
LIN {X 0,Y 118.487,Z 469.069,A -85,B 0,C 180,E1 -27207.172,E2 -27207.172} C_VEL
LIN {X 0,Y 120.153,Z 472.38,A -85,B 0,C 180,E1 -27210.358,E2 -27210.358} C_VEL
LIN {X 0,Y 121.031,Z 475.745,A -85,B 0,C 180,E1 -27212.623,E2 -27212.623} C_VEL
LIN {X 0,Y 121.133,Z 481.355,A -85,B 0,C 180,E1 -27215.284,E2 -27215.284} C_VEL
LIN {X 0,Y 120.231,Z 491.697,A -85,B 0,C 180,E1 -27219.867,E2 -27219.867} C_VEL
LIN {X 0,Y 120.281,Z 494.258,A -85,B 0,C 180,E1 -27221.358,E2 -27221.358} C_VEL
LIN {X 0,Y 120.549,Z 499.132,A -85,B 0,C 180,E1 -27224.396,E2 -27224.396} C_VEL
LIN {X 0,Y 119.023,Z 502.476,A -85,B 0,C 180,E1 -27225.503,E2 -27225.503} C_VEL
LIN {X 0,Y 113.08,Z 512.809,A -85,B 0,C 180,E1 -27229.269,E2 -27229.269} C_VEL
LIN {X 0,Y 108.1,Z 520.435,A -85,B 0,C 180,E1 -27233.037,E2 -27233.037} C_VEL
LIN {X 0,Y 102.689,Z 527.873,A -85,B 0,C 180,E1 -27237.973,E2 -27237.973} C_VEL
LIN {X 0,Y 97.387,Z 534.689,A -85,B 0,C 180,E1 -27244.347,E2 -27244.347} C_VEL
LIN {X 0,Y 93.641,Z 539.218,A -85,B 0,C 180,E1 -27250.266,E2 -27250.266} C_VEL
LIN {X 0,Y 90.564,Z 542.697,A -85,B 0,C 180,E1 -27256.543,E2 -27256.543} C_VEL
LIN {X 0,Y 89.196,Z 544.452,A -85,B 0,C 180,E1 -27260.938,E2 -27260.938} C_VEL
LIN {X 0,Y 87.985,Z 546.687,A -85,B 0,C 180,E1 -27270.005,E2 -27270.005} C_VEL
LIN {X 0,Y 88.12,Z 547.235,A -85,B 0,C 180,E1 -27274.579,E2 -27274.579} C_VEL
LIN {X 0,Y 88.498,Z 547.395,A -85,B 0,C 180,E1 -27279.144,E2 -27279.144} C_VEL
LIN {X 0,Y 89.269,Z 547.179,A -85,B 0,C 180,E1 -27283.666,E2 -27283.666} C_VEL
LIN {X 0,Y 90.861,Z 546.536,A -85,B 0,C 180,E1 -27288.028,E2 -27288.028} C_VEL
LIN {X 0,Y 93.004,Z 545.49,A -85,B 0,C 180,E1 -27292.204,E2 -27292.204} C_VEL
LIN {X 0,Y 95.443,Z 544.014,A -85,B 0,C 180,E1 -27296.225,E2 -27296.225} C_VEL
LIN {X 0,Y 99.496,Z 541.061,A -85,B 0,C 180,E1 -27302.043,E2 -27302.043} C_VEL
LIN {X 0,Y 104.31,Z 537.103,A -85,B 0,C 180,E1 -27307.333,E2 -27307.333} C_VEL
LIN {X 0,Y 109.824,Z 531.957,A -85,B 0,C 180,E1 -27312.221,E2 -27312.221} C_VEL
LIN {X 0,Y 116.005,Z 525.46,A -85,B 0,C 180,E1 -27316.641,E2 -27316.641} C_VEL
LIN {X 0,Y 122.591,Z 517.385,A -85,B 0,C 180,E1 -27320.672,E2 -27320.672} C_VEL
LIN {X 0,Y 127.328,Z 510.906,A -85,B 0,C 180,E1 -27323.025,E2 -27323.025} C_VEL
LIN {X 0,Y 127.902,Z 509.757,A -85,B 0,C 180,E1 -27323.558,E2 -27323.558} C_VEL
LIN {X 0,Y 128.016,Z 508.632,A -85,B 0,C 180,E1 -27324.378,E2 -27324.378} C_VEL
LIN {X 0,Y 127.558,Z 508.693,A -85,B 0,C 180,E1 -27324.689,E2 -27324.689} C_VEL
LIN {X 0,Y 122.296,Z 511.261,A -85,B 0,C 180,E1 -27326.91,E2 -27326.91} C_VEL
LIN {X 0,Y 112.441,Z 516.059,A -85,B 0,C 180,E1 -27332.044,E2 -27332.044} C_VEL
LIN {X 0,Y 102.386,Z 521.15,A -85,B 0,C 180,E1 -27339.926,E2 -27339.926} C_VEL
LIN {X 0,Y 96.224,Z 524.899,A -85,B 0,C 180,E1 -27347.342,E2 -27347.342} C_VEL
LIN {X 0,Y 91.306,Z 529.679,A -85,B 0,C 180,E1 -27359.999,E2 -27359.999} C_VEL
LIN {X 0,Y 90.929,Z 531.068,A -85,B 0,C 180,E1 -27364.432,E2 -27364.432} C_VEL
LIN {X 0,Y 90.574,Z 532.904,A -85,B 0,C 180,E1 -27368.927,E2 -27368.927} C_VEL
LIN {X 0,Y 94.088,Z 537.284,A -85,B 0,C 180,E1 -27381.929,E2 -27381.929} C_VEL
LIN {X 0,Y 97.256,Z 538.514,A -85,B 0,C 180,E1 -27386.269,E2 -27386.269} C_VEL
LIN {X 0,Y 105.883,Z 546.533,A -85,B 0,C 180,E1 -27394.345,E2 -27394.345} C_VEL
LIN {X 0,Y 113.638,Z 551.673,A -85,B 0,C 180,E1 -27399.518,E2 -27399.518} C_VEL
LIN {X 0,Y 112.429,Z 552.158,A -85,B 0,C 180,E1 -27401.394,E2 -27401.394} C_VEL
LIN {X 0,Y 106.251,Z 551.809,A -85,B 0,C 180,E1 -27405.841,E2 -27405.841} C_VEL
LIN {X 0,Y 99.589,Z 557.935,A -85,B 0,C 180,E1 -27410.565,E2 -27410.565} C_VEL
LIN {X 0,Y 94.258,Z 562.742,A -85,B 0,C 180,E1 -27415.994,E2 -27415.994} C_VEL
LIN {X 0,Y 90.126,Z 566.481,A -85,B 0,C 180,E1 -27422.098,E2 -27422.098} C_VEL
LIN {X 0,Y 88.1,Z 568.431,A -85,B 0,C 180,E1 -27426.488,E2 -27426.488} C_VEL
LIN {X 0,Y 85.952,Z 571.1,A -85,B 0,C 180,E1 -27435.795,E2 -27435.795} C_VEL
LIN {X 0,Y 85.786,Z 571.858,A -85,B 0,C 180,E1 -27440.565,E2 -27440.565} C_VEL
LIN {X 0,Y 86.23,Z 572.187,A -85,B 0,C 180,E1 -27445.32,E2 -27445.32} C_VEL
LIN {X 0,Y 87.056,Z 572.092,A -85,B 0,C 180,E1 -27449.995,E2 -27449.995} C_VEL
LIN {X 0,Y 86.214,Z 571.287,A -85,B 0,C 180,E1 -27454.671,E2 -27454.671} C_VEL
LIN {X 0,Y 85.745,Z 569.726,A -85,B 0,C 180,E1 -27460.407,E2 -27460.407} C_VEL
LIN {X 0,Y 86.449,Z 566.216,A -85,B 0,C 180,E1 -27468.971,E2 -27468.971} C_VEL
LIN {X 0,Y 88.526,Z 562.156,A -85,B 0,C 180,E1 -27475.884,E2 -27475.884} C_VEL
LIN {X 0,Y 92.441,Z 556.129,A -85,B 0,C 180,E1 -27483.251,E2 -27483.251} C_VEL
LIN {X 0,Y 97.216,Z 549.212,A -85,B 0,C 180,E1 -27489.233,E2 -27489.233} C_VEL
LIN {X 0,Y 99.732,Z 545.215,A -85,B 0,C 180,E1 -27492.018,E2 -27492.018} C_VEL
LIN {X 0,Y 104.143,Z 535.524,A -85,B 0,C 180,E1 -27497.923,E2 -27497.923} C_VEL
LIN {X 0,Y 108.626,Z 525.532,A -85,B 0,C 180,E1 -27502.418,E2 -27502.418} C_VEL
LIN {X 0,Y 113.251,Z 514.166,A -85,B 0,C 180,E1 -27506.295,E2 -27506.295} C_VEL
LIN {X 0,Y 117.018,Z 503.39,A -85,B 0,C 180,E1 -27509.102,E2 -27509.102} C_VEL
LIN {X 0,Y 118.589,Z 496.258,A -85,B 0,C 180,E1 -27510.974,E2 -27510.974} C_VEL
LIN {X 0,Y 119.035,Z 493.287,A -85,B 0,C 180,E1 -27511.815,E2 -27511.815} C_VEL
LIN {X 0,Y 117.657,Z 484.436,A -85,B 0,C 180,E1 -27516.223,E2 -27516.223} C_VEL
LIN {X 0,Y 116.998,Z 481.476,A -85,B 0,C 180,E1 -27517.95,E2 -27517.95} C_VEL
LIN {X 0,Y 113.829,Z 474.776,A -85,B 0,C 180,E1 -27524.329,E2 -27524.329} C_VEL
LIN {X 0,Y 111.153,Z 469.394,A -85,B 0,C 180,E1 -27532.051,E2 -27532.051} C_VEL
LIN {X 0,Y 110.041,Z 465.851,A -85,B 0,C 180,E1 -27540.001,E2 -27540.001} C_VEL
LIN {X 0,Y 109.913,Z 465.825,A -85,B 0,C 180,E1 -27545.505,E2 -27545.505} C_VEL
LIN {X 0,Y 110.642,Z 466.714,A -85,B 0,C 180,E1 -27551.45,E2 -27551.45} C_VEL
LIN {X 0,Y 111.28,Z 467.877,A -85,B 0,C 180,E1 -27554.634,E2 -27554.634} C_VEL
LIN {X 0,Y 113.533,Z 471.642,A -85,B 0,C 180,E1 -27561.804,E2 -27561.804} C_VEL
LIN {X 0,Y 115.915,Z 476.652,A -85,B 0,C 180,E1 -27567.827,E2 -27567.827} C_VEL
LIN {X 0,Y 117.429,Z 480.667,A -85,B 0,C 180,E1 -27571.581,E2 -27571.581} C_VEL
LIN {X 0,Y 119.028,Z 486.602,A -85,B 0,C 180,E1 -27576.19,E2 -27576.19} C_VEL
LIN {X 0,Y 120.157,Z 492.934,A -85,B 0,C 180,E1 -27580.509,E2 -27580.509} C_VEL
LIN {X 0,Y 120.281,Z 494.258,A -85,B 0,C 180,E1 -27581.358,E2 -27581.358} C_VEL
LIN {X 0,Y 119.882,Z 496.544,A -85,B 0,C 180,E1 -27582.405,E2 -27582.405} C_VEL
LIN {X 0,Y 117.992,Z 500.212,A -85,B 0,C 180,E1 -27583.366,E2 -27583.366} C_VEL
LIN {X 0,Y 111.394,Z 508.797,A -85,B 0,C 180,E1 -27584.887,E2 -27584.887} C_VEL
LIN {X 0,Y 109.922,Z 510.851,A -85,B 0,C 180,E1 -27585.558,E2 -27585.558} C_VEL
LIN {X 0,Y 104.648,Z 518.722,A -85,B 0,C 180,E1 -27589.102,E2 -27589.102} C_VEL
LIN {X 0,Y 98.696,Z 526.681,A -85,B 0,C 180,E1 -27594.028,E2 -27594.028} C_VEL
LIN {X 0,Y 94.219,Z 532.122,A -85,B 0,C 180,E1 -27598.53,E2 -27598.53} C_VEL
LIN {X 0,Y 89.65,Z 537.406,A -85,B 0,C 180,E1 -27604.464,E2 -27604.464} C_VEL
LIN {X 0,Y 85.905,Z 541.538,A -85,B 0,C 180,E1 -27610.904,E2 -27610.904} C_VEL
LIN {X 0,Y 83.749,Z 543.757,A -85,B 0,C 180,E1 -27615.424,E2 -27615.424} C_VEL
LIN {X 0,Y 82.265,Z 545.495,A -85,B 0,C 180,E1 -27620.168,E2 -27620.168} C_VEL
LIN {X 0,Y 80.957,Z 547.713,A -85,B 0,C 180,E1 -27630.005,E2 -27630.005} C_VEL
LIN {X 0,Y 81.115,Z 548.25,A -85,B 0,C 180,E1 -27634.976,E2 -27634.976} C_VEL
LIN {X 0,Y 81.564,Z 548.396,A -85,B 0,C 180,E1 -27639.929,E2 -27639.929} C_VEL
LIN {X 0,Y 82.451,Z 548.17,A -85,B 0,C 180,E1 -27644.821,E2 -27644.821} C_VEL
LIN {X 0,Y 84.202,Z 547.519,A -85,B 0,C 180,E1 -27649.509,E2 -27649.509} C_VEL
LIN {X 0,Y 86.536,Z 546.458,A -85,B 0,C 180,E1 -27653.964,E2 -27653.964} C_VEL
LIN {X 0,Y 89.188,Z 544.971,A -85,B 0,C 180,E1 -27658.221,E2 -27658.221} C_VEL
LIN {X 0,Y 93.58,Z 542.018,A -85,B 0,C 180,E1 -27664.296,E2 -27664.296} C_VEL
LIN {X 0,Y 98.783,Z 538.024,A -85,B 0,C 180,E1 -27669.82,E2 -27669.82} C_VEL
LIN {X 0,Y 105.78,Z 531.882,A -85,B 0,C 180,E1 -27675.585,E2 -27675.585} C_VEL
LIN {X 0,Y 112.404,Z 525.108,A -85,B 0,C 180,E1 -27679.994,E2 -27679.994} C_VEL
LIN {X 0,Y 118.95,Z 517.318,A -85,B 0,C 180,E1 -27683.665,E2 -27683.665} C_VEL
LIN {X 0,Y 119.753,Z 516.295,A -85,B 0,C 180,E1 -27684.063,E2 -27684.063} C_VEL
LIN {X 0,Y 115.173,Z 517.772,A -85,B 0,C 180,E1 -27686.687,E2 -27686.687} C_VEL
LIN {X 0,Y 110.01,Z 520.152,A -85,B 0,C 180,E1 -27689.263,E2 -27689.263} C_VEL
LIN {X 0,Y 97.215,Z 526.024,A -85,B 0,C 180,E1 -27698.809,E2 -27698.809} C_VEL
LIN {X 0,Y 90.825,Z 529.621,A -85,B 0,C 180,E1 -27706.576,E2 -27706.576} C_VEL
LIN {X 0,Y 84.965,Z 536.516,A -85,B 0,C 180,E1 -27726.937,E2 -27726.937} C_VEL
LIN {X 0,Y 88.869,Z 541.575,A -85,B 0,C 180,E1 -27743.291,E2 -27743.291} C_VEL
LIN {X 0,Y 91.674,Z 542.606,A -85,B 0,C 180,E1 -27747.385,E2 -27747.385} C_VEL
LIN {X 0,Y 94.362,Z 544.092,A -85,B 0,C 180,E1 -27751.422,E2 -27751.422} C_VEL
LIN {X 0,Y 99.016,Z 545.365,A -85,B 0,C 180,E1 -27755.842,E2 -27755.842} C_VEL
LIN {X 0,Y 100.139,Z 545.52,A -85,B 0,C 180,E1 -27756.622,E2 -27756.622} C_VEL
LIN {X 0,Y 104.175,Z 548.358,A -85,B 0,C 180,E1 -27759.4,E2 -27759.4} C_VEL
LIN {X 0,Y 104.625,Z 549.248,A -85,B 0,C 180,E1 -27761.045,E2 -27761.045} C_VEL
LIN {X 0,Y 103.184,Z 549.238,A -85,B 0,C 180,E1 -27762.02,E2 -27762.02} C_VEL
LIN {X 0,Y 96.404,Z 555.173,A -85,B 0,C 180,E1 -27766.161,E2 -27766.161} C_VEL
LIN {X 0,Y 90.253,Z 560.32,A -85,B 0,C 180,E1 -27771.462,E2 -27771.462} C_VEL
LIN {X 0,Y 85.232,Z 564.374,A -85,B 0,C 180,E1 -27777.584,E2 -27777.584} C_VEL
LIN {X 0,Y 81.583,Z 567.445,A -85,B 0,C 180,E1 -27784.481,E2 -27784.481} C_VEL
LIN {X 0,Y 79.018,Z 570.096,A -85,B 0,C 180,E1 -27794.519,E2 -27794.519} C_VEL
LIN {X 0,Y 78.75,Z 570.847,A -85,B 0,C 180,E1 -27799.713,E2 -27799.713} C_VEL
LIN {X 0,Y 79.111,Z 571.161,A -85,B 0,C 180,E1 -27804.898,E2 -27804.898} C_VEL
LIN {X 0,Y 79.924,Z 571.06,A -85,B 0,C 180,E1 -27809.995,E2 -27809.995} C_VEL
LIN {X 0,Y 79.083,Z 570.244,A -85,B 0,C 180,E1 -27815.093,E2 -27815.093} C_VEL
LIN {X 0,Y 78.672,Z 568.865,A -85,B 0,C 180,E1 -27820.692,E2 -27820.692} C_VEL
LIN {X 0,Y 79.65,Z 565.129,A -85,B 0,C 180,E1 -27830.661,E2 -27830.661} C_VEL
LIN {X 0,Y 82.081,Z 561.05,A -85,B 0,C 180,E1 -27838.088,E2 -27838.088} C_VEL
LIN {X 0,Y 86.082,Z 555.55,A -85,B 0,C 180,E1 -27845.272,E2 -27845.272} C_VEL
LIN {X 0,Y 91.749,Z 548.057,A -85,B 0,C 180,E1 -27852.08,E2 -27852.08} C_VEL
LIN {X 0,Y 93.509,Z 545.437,A -85,B 0,C 180,E1 -27854.037,E2 -27854.037} C_VEL
LIN {X 0,Y 98.382,Z 535.919,A -85,B 0,C 180,E1 -27860.247,E2 -27860.247} C_VEL
LIN {X 0,Y 103.168,Z 526.432,A -85,B 0,C 180,E1 -27864.823,E2 -27864.823} C_VEL
LIN {X 0,Y 107.901,Z 516.041,A -85,B 0,C 180,E1 -27868.597,E2 -27868.597} C_VEL
LIN {X 0,Y 112.442,Z 504.516,A -85,B 0,C 180,E1 -27871.754,E2 -27871.754} C_VEL
LIN {X 0,Y 114.118,Z 498.304,A -85,B 0,C 180,E1 -27873.482,E2 -27873.482} C_VEL
LIN {X 0,Y 114.492,Z 496.402,A -85,B 0,C 180,E1 -27874.065,E2 -27874.065} C_VEL
LIN {X 0,Y 113.699,Z 488.803,A -85,B 0,C 180,E1 -27878.231,E2 -27878.231} C_VEL
LIN {X 0,Y 113.129,Z 486.256,A -85,B 0,C 180,E1 -27880.022,E2 -27880.022} C_VEL
LIN {X 0,Y 111.039,Z 481.006,A -85,B 0,C 180,E1 -27885.336,E2 -27885.336} C_VEL
LIN {X 0,Y 108.807,Z 475.576,A -85,B 0,C 180,E1 -27893.511,E2 -27893.511} C_VEL
LIN {X 0,Y 108.114,Z 472.778,A -85,B 0,C 180,E1 -27900.001,E2 -27900.001} C_VEL
LIN {X 0,Y 107.95,Z 472.501,A -85,B 0,C 180,E1 -27903.734,E2 -27903.734} C_VEL
LIN {X 0,Y 108.443,Z 473.445,A -85,B 0,C 180,E1 -27911.212,E2 -27911.212} C_VEL
LIN {X 0,Y 109.025,Z 474.888,A -85,B 0,C 180,E1 -27914.944,E2 -27914.944} C_VEL
LIN {X 0,Y 110.582,Z 477.962,A -85,B 0,C 180,E1 -27921.093,E2 -27921.093} C_VEL
LIN {X 0,Y 112.044,Z 481.741,A -85,B 0,C 180,E1 -27926.046,E2 -27926.046} C_VEL
LIN {X 0,Y 113.175,Z 485.295,A -85,B 0,C 180,E1 -27929.789,E2 -27929.789} C_VEL
LIN {X 0,Y 114.416,Z 491.317,A -85,B 0,C 180,E1 -27934.898,E2 -27934.898} C_VEL
LIN {X 0,Y 115.074,Z 497.079,A -85,B 0,C 180,E1 -27939.209,E2 -27939.209} C_VEL
LIN {X 0,Y 115.164,Z 501.394,A -85,B 0,C 180,E1 -27942.168,E2 -27942.168} C_VEL
LIN {X 0,Y 114.73,Z 502.631,A -85,B 0,C 180,E1 -27942.692,E2 -27942.692} C_VEL
LIN {X 0,Y 109.922,Z 510.851,A -85,B 0,C 180,E1 -27945.558,E2 -27945.558} C_VEL
LIN {X 0,Y 106.744,Z 515.078,A -85,B 0,C 180,E1 -27947.032,E2 -27947.032} C_VEL
LIN {X 0,Y 97.563,Z 524.083,A -85,B 0,C 180,E1 -27949.957,E2 -27949.957} C_VEL
LIN {X 0,Y 92.523,Z 528.722,A -85,B 0,C 180,E1 -27952.308,E2 -27952.308} C_VEL
LIN {X 0,Y 90.49,Z 530.829,A -85,B 0,C 180,E1 -27953.928,E2 -27953.928} C_VEL
LIN {X 0,Y 84.954,Z 536.886,A -85,B 0,C 180,E1 -27960.247,E2 -27960.247} C_VEL
LIN {X 0,Y 80.575,Z 541.373,A -85,B 0,C 180,E1 -27966.896,E2 -27966.896} C_VEL
LIN {X 0,Y 76.971,Z 544.818,A -85,B 0,C 180,E1 -27974.108,E2 -27974.108} C_VEL
LIN {X 0,Y 75.352,Z 546.537,A -85,B 0,C 180,E1 -27979.255,E2 -27979.255} C_VEL
LIN {X 0,Y 73.929,Z 548.739,A -85,B 0,C 180,E1 -27990.006,E2 -27990.006} C_VEL
LIN {X 0,Y 74.115,Z 549.263,A -85,B 0,C 180,E1 -27995.447,E2 -27995.447} C_VEL
LIN {X 0,Y 74.648,Z 549.396,A -85,B 0,C 180,E1 -28000.859,E2 -28000.859} C_VEL
LIN {X 0,Y 75.673,Z 549.162,A -85,B 0,C 180,E1 -28006.184,E2 -28006.184} C_VEL
LIN {X 0,Y 77.609,Z 548.502,A -85,B 0,C 180,E1 -28011.243,E2 -28011.243} C_VEL
LIN {X 0,Y 80.163,Z 547.424,A -85,B 0,C 180,E1 -28016.005,E2 -28016.005} C_VEL
LIN {X 0,Y 83.057,Z 545.927,A -85,B 0,C 180,E1 -28020.517,E2 -28020.517} C_VEL
LIN {X 0,Y 87.837,Z 542.97,A -85,B 0,C 180,E1 -28026.856,E2 -28026.856} C_VEL
LIN {X 0,Y 93.467,Z 538.944,A -85,B 0,C 180,E1 -28032.594,E2 -28032.594} C_VEL
LIN {X 0,Y 100.966,Z 532.779,A -85,B 0,C 180,E1 -28038.448,E2 -28038.448} C_VEL
LIN {X 0,Y 108.01,Z 525.965,A -85,B 0,C 180,E1 -28042.858,E2 -28042.858} C_VEL
LIN {X 0,Y 109.211,Z 524.662,A -85,B 0,C 180,E1 -28043.559,E2 -28043.559} C_VEL
LIN {X 0,Y 110.336,Z 522.856,A -85,B 0,C 180,E1 -28045.02,E2 -28045.02} C_VEL
LIN {X 0,Y 95.822,Z 528.816,A -85,B 0,C 180,E1 -28053.89,E2 -28053.89} C_VEL
LIN {X 0,Y 85.165,Z 533.981,A -85,B 0,C 180,E1 -28065.665,E2 -28065.665} C_VEL
LIN {X 0,Y 79.166,Z 541.51,A -85,B 0,C 180,E1 -28090.226,E2 -28090.226} C_VEL
LIN {X 0,Y 83.476,Z 545.549,A -85,B 0,C 180,E1 -28104.894,E2 -28104.894} C_VEL
LIN {X 0,Y 86.38,Z 546.644,A -85,B 0,C 180,E1 -28109.219,E2 -28109.219} C_VEL
LIN {X 0,Y 89.332,Z 548.051,A -85,B 0,C 180,E1 -28113.414,E2 -28113.414} C_VEL
LIN {X 0,Y 95.069,Z 549.434,A -85,B 0,C 180,E1 -28118.522,E2 -28118.522} C_VEL
LIN {X 0,Y 95.842,Z 550.666,A -85,B 0,C 180,E1 -28120.383,E2 -28120.383} C_VEL
LIN {X 0,Y 89.102,Z 556.1,A -85,B 0,C 180,E1 -28124.768,E2 -28124.768} C_VEL
LIN {X 0,Y 82.85,Z 560.858,A -85,B 0,C 180,E1 -28130.484,E2 -28130.484} C_VEL
LIN {X 0,Y 77.764,Z 564.547,A -85,B 0,C 180,E1 -28137.156,E2 -28137.156} C_VEL
LIN {X 0,Y 75.183,Z 566.46,A -85,B 0,C 180,E1 -28142.129,E2 -28142.129} C_VEL
LIN {X 0,Y 72.142,Z 569.093,A -85,B 0,C 180,E1 -28153.001,E2 -28153.001} C_VEL
LIN {X 0,Y 71.713,Z 569.831,A -85,B 0,C 180,E1 -28158.691,E2 -28158.691} C_VEL
LIN {X 0,Y 71.987,Z 570.135,A -85,B 0,C 180,E1 -28164.391,E2 -28164.391} C_VEL
LIN {X 0,Y 72.787,Z 570.028,A -85,B 0,C 180,E1 -28169.994,E2 -28169.994} C_VEL
LIN {X 0,Y 71.956,Z 569.201,A -85,B 0,C 180,E1 -28175.599,E2 -28175.599} C_VEL
LIN {X 0,Y 71.624,Z 567.928,A -85,B 0,C 180,E1 -28181.311,E2 -28181.311} C_VEL
LIN {X 0,Y 72.354,Z 565.196,A -85,B 0,C 180,E1 -28189.868,E2 -28189.868} C_VEL
LIN {X 0,Y 74.677,Z 561.451,A -85,B 0,C 180,E1 -28198.064,E2 -28198.064} C_VEL
LIN {X 0,Y 78.422,Z 556.699,A -85,B 0,C 180,E1 -28205.45,E2 -28205.45} C_VEL
LIN {X 0,Y 83.61,Z 550.491,A -85,B 0,C 180,E1 -28212.249,E2 -28212.249} C_VEL
LIN {X 0,Y 87.411,Z 545.599,A -85,B 0,C 180,E1 -28216.346,E2 -28216.346} C_VEL
LIN {X 0,Y 92.473,Z 536.833,A -85,B 0,C 180,E1 -28222.556,E2 -28222.556} C_VEL
LIN {X 0,Y 97.905,Z 527.191,A -85,B 0,C 180,E1 -28227.498,E2 -28227.498} C_VEL
LIN {X 0,Y 103.442,Z 516.338,A -85,B 0,C 180,E1 -28231.603,E2 -28231.603} C_VEL
LIN {X 0,Y 108.61,Z 504.352,A -85,B 0,C 180,E1 -28234.937,E2 -28234.937} C_VEL
LIN {X 0,Y 109.948,Z 499.726,A -85,B 0,C 180,E1 -28236.36,E2 -28236.36} C_VEL
LIN {X 0,Y 109.688,Z 493.057,A -85,B 0,C 180,E1 -28240.344,E2 -28240.344} C_VEL
LIN {X 0,Y 109.477,Z 491.851,A -85,B 0,C 180,E1 -28241.279,E2 -28241.279} C_VEL
LIN {X 0,Y 107.807,Z 486.76,A -85,B 0,C 180,E1 -28246.812,E2 -28246.812} C_VEL
LIN {X 0,Y 106.503,Z 483.074,A -85,B 0,C 180,E1 -28252.417,E2 -28252.417} C_VEL
LIN {X 0,Y 105.783,Z 479.646,A -85,B 0,C 180,E1 -28260.001,E2 -28260.001} C_VEL
LIN {X 0,Y 105.624,Z 479.198,A -85,B 0,C 180,E1 -28263.816,E2 -28263.816} C_VEL
LIN {X 0,Y 105.627,Z 479.505,A -85,B 0,C 180,E1 -28267.648,E2 -28267.648} C_VEL
LIN {X 0,Y 105.921,Z 480.262,A -85,B 0,C 180,E1 -28271.483,E2 -28271.483} C_VEL
LIN {X 0,Y 107.047,Z 483.555,A -85,B 0,C 180,E1 -28279.165,E2 -28279.165} C_VEL
LIN {X 0,Y 107.856,Z 485.954,A -85,B 0,C 180,E1 -28283.016,E2 -28283.016} C_VEL
LIN {X 0,Y 108.972,Z 490.133,A -85,B 0,C 180,E1 -28288.161,E2 -28288.161} C_VEL
LIN {X 0,Y 109.607,Z 494.446,A -85,B 0,C 180,E1 -28292.277,E2 -28292.277} C_VEL
LIN {X 0,Y 109.96,Z 500.762,A -85,B 0,C 180,E1 -28297.49,E2 -28297.49} C_VEL
LIN {X 0,Y 109.889,Z 503.912,A -85,B 0,C 180,E1 -28299.88,E2 -28299.88} C_VEL
LIN {X 0,Y 107.718,Z 507.875,A -85,B 0,C 180,E1 -28301.333,E2 -28301.333} C_VEL
LIN {X 0,Y 101.683,Z 516.796,A -85,B 0,C 180,E1 -28304.898,E2 -28304.898} C_VEL
LIN {X 0,Y 95.15,Z 525.367,A -85,B 0,C 180,E1 -28309.744,E2 -28309.744} C_VEL
LIN {X 0,Y 90.49,Z 530.829,A -85,B 0,C 180,E1 -28313.928,E2 -28313.928} C_VEL
LIN {X 0,Y 87.337,Z 533.878,A -85,B 0,C 180,E1 -28316.483,E2 -28316.483} C_VEL
LIN {X 0,Y 80.855,Z 538.513,A -85,B 0,C 180,E1 -28320.504,E2 -28320.504} C_VEL
LIN {X 0,Y 74.552,Z 542.548,A -85,B 0,C 180,E1 -28325.354,E2 -28325.354} C_VEL
LIN {X 0,Y 71.858,Z 544.503,A -85,B 0,C 180,E1 -28329.172,E2 -28329.172} C_VEL
LIN {X 0,Y 68.463,Z 547.58,A -85,B 0,C 180,E1 -28338.159,E2 -28338.159} C_VEL
LIN {X 0,Y 66.901,Z 549.764,A -85,B 0,C 180,E1 -28350.007,E2 -28350.007} C_VEL
LIN {X 0,Y 67.12,Z 550.275,A -85,B 0,C 180,E1 -28356.017,E2 -28356.017} C_VEL
LIN {X 0,Y 68.945,Z 550.155,A -85,B 0,C 180,E1 -28367.813,E2 -28367.813} C_VEL
LIN {X 0,Y 71.1,Z 549.485,A -85,B 0,C 180,E1 -28373.296,E2 -28373.296} C_VEL
LIN {X 0,Y 73.909,Z 548.389,A -85,B 0,C 180,E1 -28378.395,E2 -28378.395} C_VEL
LIN {X 0,Y 77.08,Z 546.884,A -85,B 0,C 180,E1 -28383.172,E2 -28383.172} C_VEL
LIN {X 0,Y 82.298,Z 543.919,A -85,B 0,C 180,E1 -28389.772,E2 -28389.772} C_VEL
LIN {X 0,Y 88.398,Z 539.865,A -85,B 0,C 180,E1 -28395.694,E2 -28395.694} C_VEL
LIN {X 0,Y 96.432,Z 533.675,A -85,B 0,C 180,E1 -28401.586,E2 -28401.586} C_VEL
LIN {X 0,Y 100.13,Z 530.445,A -85,B 0,C 180,E1 -28403.827,E2 -28403.827} C_VEL
LIN {X 0,Y 101.234,Z 528.969,A -85,B 0,C 180,E1 -28405.278,E2 -28405.278} C_VEL
LIN {X 0,Y 86.286,Z 534.754,A -85,B 0,C 180,E1 -28415.966,E2 -28415.966} C_VEL
LIN {X 0,Y 76.836,Z 539.468,A -85,B 0,C 180,E1 -28429.458,E2 -28429.458} C_VEL
LIN {X 0,Y 74.061,Z 546.607,A -85,B 0,C 180,E1 -28456.539,E2 -28456.539} C_VEL
LIN {X 0,Y 77.966,Z 549.2,A -85,B 0,C 180,E1 -28466.788,E2 -28466.788} C_VEL
LIN {X 0,Y 86.977,Z 552.38,A -85,B 0,C 180,E1 -28478.323,E2 -28478.323} C_VEL
LIN {X 0,Y 86.03,Z 553.86,A -85,B 0,C 180,E1 -28480.128,E2 -28480.128} C_VEL
LIN {X 0,Y 79.608,Z 558.435,A -85,B 0,C 180,E1 -28485.061,E2 -28485.061} C_VEL
LIN {X 0,Y 73.588,Z 562.447,A -85,B 0,C 180,E1 -28491.62,E2 -28491.62} C_VEL
LIN {X 0,Y 68.936,Z 565.475,A -85,B 0,C 180,E1 -28499.346,E2 -28499.346} C_VEL
LIN {X 0,Y 65.325,Z 568.091,A -85,B 0,C 180,E1 -28511.164,E2 -28511.164} C_VEL
LIN {X 0,Y 64.719,Z 568.837,A -85,B 0,C 180,E1 -28517.772,E2 -28517.772} C_VEL
LIN {X 0,Y 64.875,Z 569.109,A -85,B 0,C 180,E1 -28523.774,E2 -28523.774} C_VEL
LIN {X 0,Y 65.646,Z 568.995,A -85,B 0,C 180,E1 -28529.993,E2 -28529.993} C_VEL
LIN {X 0,Y 64.814,Z 568.154,A -85,B 0,C 180,E1 -28536.218,E2 -28536.218} C_VEL
LIN {X 0,Y 64.576,Z 566.861,A -85,B 0,C 180,E1 -28542.565,E2 -28542.565} C_VEL
LIN {X 0,Y 66.362,Z 562.96,A -85,B 0,C 180,E1 -28555.055,E2 -28555.055} C_VEL
LIN {X 0,Y 69.694,Z 558.843,A -85,B 0,C 180,E1 -28563.677,E2 -28563.677} C_VEL
LIN {X 0,Y 74.555,Z 553.594,A -85,B 0,C 180,E1 -28571.281,E2 -28571.281} C_VEL
LIN {X 0,Y 80.53,Z 547.011,A -85,B 0,C 180,E1 -28577.877,E2 -28577.877} C_VEL
LIN {X 0,Y 86.2,Z 538.479,A -85,B 0,C 180,E1 -28584.609,E2 -28584.609} C_VEL
LIN {X 0,Y 91.735,Z 529.865,A -85,B 0,C 180,E1 -28589.518,E2 -28589.518} C_VEL
LIN {X 0,Y 97.277,Z 520.316,A -85,B 0,C 180,E1 -28593.586,E2 -28593.586} C_VEL
LIN {X 0,Y 102.829,Z 509.396,A -85,B 0,C 180,E1 -28597.009,E2 -28597.009} C_VEL
LIN {X 0,Y 104.815,Z 504.84,A -85,B 0,C 180,E1 -28598.243,E2 -28598.243} C_VEL
LIN {X 0,Y 105.466,Z 502.855,A -85,B 0,C 180,E1 -28598.883,E2 -28598.883} C_VEL
LIN {X 0,Y 105.651,Z 498.618,A -85,B 0,C 180,E1 -28601.581,E2 -28601.581} C_VEL
LIN {X 0,Y 105.577,Z 497.313,A -85,B 0,C 180,E1 -28602.57,E2 -28602.57} C_VEL
LIN {X 0,Y 104.746,Z 493.823,A -85,B 0,C 180,E1 -28606.419,E2 -28606.419} C_VEL
LIN {X 0,Y 103.613,Z 489.938,A -85,B 0,C 180,E1 -28612.204,E2 -28612.204} C_VEL
LIN {X 0,Y 103.031,Z 486.324,A -85,B 0,C 180,E1 -28620.001,E2 -28620.001} C_VEL
LIN {X 0,Y 102.896,Z 485.759,A -85,B 0,C 180,E1 -28623.917,E2 -28623.917} C_VEL
LIN {X 0,Y 102.835,Z 486.095,A -85,B 0,C 180,E1 -28627.857,E2 -28627.857} C_VEL
LIN {X 0,Y 103.004,Z 486.978,A -85,B 0,C 180,E1 -28631.813,E2 -28631.813} C_VEL
LIN {X 0,Y 103.838,Z 490.319,A -85,B 0,C 180,E1 -28639.781,E2 -28639.781} C_VEL
LIN {X 0,Y 104.606,Z 494.171,A -85,B 0,C 180,E1 -28645.514,E2 -28645.514} C_VEL
LIN {X 0,Y 104.973,Z 499.175,A -85,B 0,C 180,E1 -28650.905,E2 -28650.905} C_VEL
LIN {X 0,Y 104.903,Z 504.114,A -85,B 0,C 180,E1 -28655.388,E2 -28655.388} C_VEL
LIN {X 0,Y 104.73,Z 506.189,A -85,B 0,C 180,E1 -28657.155,E2 -28657.155} C_VEL
LIN {X 0,Y 103.883,Z 508.061,A -85,B 0,C 180,E1 -28658.068,E2 -28658.068} C_VEL
LIN {X 0,Y 98.104,Z 516.368,A -85,B 0,C 180,E1 -28661.226,E2 -28661.226} C_VEL
LIN {X 0,Y 91.005,Z 525.209,A -85,B 0,C 180,E1 -28665.977,E2 -28665.977} C_VEL
LIN {X 0,Y 84.599,Z 532.302,A -85,B 0,C 180,E1 -28671.468,E2 -28671.468} C_VEL
LIN {X 0,Y 78.938,Z 537.984,A -85,B 0,C 180,E1 -28677.718,E2 -28677.718} C_VEL
LIN {X 0,Y 74.174,Z 542.45,A -85,B 0,C 180,E1 -28684.769,E2 -28684.769} C_VEL
LIN {X 0,Y 71.858,Z 544.503,A -85,B 0,C 180,E1 -28689.172,E2 -28689.172} C_VEL
LIN {X 0,Y 69.433,Z 546.261,A -85,B 0,C 180,E1 -28693.302,E2 -28693.302} C_VEL
LIN {X 0,Y 64.486,Z 548.739,A -85,B 0,C 180,E1 -28700.352,E2 -28700.352} C_VEL
LIN {X 0,Y 60.581,Z 550.539,A -85,B 0,C 180,E1 -28708.558,E2 -28708.558} C_VEL
LIN {X 0,Y 59.934,Z 551.092,A -85,B 0,C 180,E1 -28714.112,E2 -28714.112} C_VEL
LIN {X 0,Y 60.895,Z 551.396,A -85,B 0,C 180,E1 -28723.353,E2 -28723.353} C_VEL
LIN {X 0,Y 62.286,Z 551.147,A -85,B 0,C 180,E1 -28729.793,E2 -28729.793} C_VEL
LIN {X 0,Y 64.702,Z 550.469,A -85,B 0,C 180,E1 -28735.76,E2 -28735.76} C_VEL
LIN {X 0,Y 67.806,Z 549.355,A -85,B 0,C 180,E1 -28741.221,E2 -28741.221} C_VEL
LIN {X 0,Y 71.296,Z 547.841,A -85,B 0,C 180,E1 -28746.267,E2 -28746.267} C_VEL
LIN {X 0,Y 76.938,Z 544.903,A -85,B 0,C 180,E1 -28753.047,E2 -28753.047} C_VEL
LIN {X 0,Y 83.62,Z 540.786,A -85,B 0,C 180,E1 -28759.157,E2 -28759.157} C_VEL
LIN {X 0,Y 90.203,Z 536.118,A -85,B 0,C 180,E1 -28763.761,E2 -28763.761} C_VEL
LIN {X 0,Y 91.393,Z 534.709,A -85,B 0,C 180,E1 -28765.883,E2 -28765.883} C_VEL
LIN {X 0,Y 76.634,Z 540.164,A -85,B 0,C 180,E1 -28778.478,E2 -28778.478} C_VEL
LIN {X 0,Y 66.922,Z 548.688,A -85,B 0,C 180,E1 -28812.123,E2 -28812.123} C_VEL
LIN {X 0,Y 72.363,Z 552.516,A -85,B 0,C 180,E1 -28829.051,E2 -28829.051} C_VEL
LIN {X 0,Y 78.134,Z 554.593,A -85,B 0,C 180,E1 -28837.243,E2 -28837.243} C_VEL
LIN {X 0,Y 77.198,Z 555.931,A -85,B 0,C 180,E1 -28839.297,E2 -28839.297} C_VEL
LIN {X 0,Y 70.212,Z 560.269,A -85,B 0,C 180,E1 -28845.51,E2 -28845.51} C_VEL
LIN {X 0,Y 66.23,Z 562.615,A -85,B 0,C 180,E1 -28850.446,E2 -28850.446} C_VEL
LIN {X 0,Y 62.887,Z 564.491,A -85,B 0,C 180,E1 -28856.02,E2 -28856.02} C_VEL
LIN {X 0,Y 58.592,Z 567.088,A -85,B 0,C 180,E1 -28868.902,E2 -28868.902} C_VEL
LIN {X 0,Y 57.746,Z 567.851,A -85,B 0,C 180,E1 -28876.807,E2 -28876.807} C_VEL
LIN {X 0,Y 58.498,Z 567.961,A -85,B 0,C 180,E1 -28889.993,E2 -28889.993} C_VEL
LIN {X 0,Y 57.529,Z 566.182,A -85,B 0,C 180,E1 -28902.234,E2 -28902.234} C_VEL
LIN {X 0,Y 58.98,Z 563.023,A -85,B 0,C 180,E1 -28914.641,E2 -28914.641} C_VEL
LIN {X 0,Y 62.324,Z 559.243,A -85,B 0,C 180,E1 -28924.312,E2 -28924.312} C_VEL
LIN {X 0,Y 68.106,Z 553.589,A -85,B 0,C 180,E1 -28933.753,E2 -28933.753} C_VEL
LIN {X 0,Y 74.719,Z 547.047,A -85,B 0,C 180,E1 -28940.885,E2 -28940.885} C_VEL
LIN {X 0,Y 80.92,Z 538.816,A -85,B 0,C 180,E1 -28947.854,E2 -28947.854} C_VEL
LIN {X 0,Y 86.892,Z 530.468,A -85,B 0,C 180,E1 -28952.824,E2 -28952.824} C_VEL
LIN {X 0,Y 92.89,Z 521.138,A -85,B 0,C 180,E1 -28956.907,E2 -28956.907} C_VEL
LIN {X 0,Y 98.49,Z 511.246,A -85,B 0,C 180,E1 -28960.09,E2 -28960.09} C_VEL
LIN {X 0,Y 100.399,Z 507.483,A -85,B 0,C 180,E1 -28961.096,E2 -28961.096} C_VEL
LIN {X 0,Y 101.091,Z 505.674,A -85,B 0,C 180,E1 -28961.768,E2 -28961.768} C_VEL
LIN {X 0,Y 101.436,Z 502.623,A -85,B 0,C 180,E1 -28963.911,E2 -28963.911} C_VEL
LIN {X 0,Y 100.89,Z 499.19,A -85,B 0,C 180,E1 -28967.938,E2 -28967.938} C_VEL
LIN {X 0,Y 100.122,Z 495.544,A -85,B 0,C 180,E1 -28973.957,E2 -28973.957} C_VEL
LIN {X 0,Y 99.903,Z 492.851,A -85,B 0,C 180,E1 -28980.001,E2 -28980.001} C_VEL
LIN {X 0,Y 99.812,Z 492.167,A -85,B 0,C 180,E1 -28984.039,E2 -28984.039} C_VEL
LIN {X 0,Y 99.646,Z 492.766,A -85,B 0,C 180,E1 -28989.131,E2 -28989.131} C_VEL
LIN {X 0,Y 99.653,Z 493.514,A -85,B 0,C 180,E1 -28992.216,E2 -28992.216} C_VEL
LIN {X 0,Y 100.049,Z 496.131,A -85,B 0,C 180,E1 -28998.953,E2 -28998.953} C_VEL
LIN {X 0,Y 100.368,Z 499.837,A -85,B 0,C 180,E1 -29004.844,E2 -29004.844} C_VEL
LIN {X 0,Y 100.269,Z 503.738,A -85,B 0,C 180,E1 -29009.384,E2 -29009.384} C_VEL
LIN {X 0,Y 99.743,Z 508.706,A -85,B 0,C 180,E1 -29014.313,E2 -29014.313} C_VEL
LIN {X 0,Y 98.971,Z 510.361,A -85,B 0,C 180,E1 -29015.269,E2 -29015.269} C_VEL
LIN {X 0,Y 92.339,Z 519.13,A -85,B 0,C 180,E1 -29018.736,E2 -29018.736} C_VEL
LIN {X 0,Y 84.935,Z 527.652,A -85,B 0,C 180,E1 -29023.621,E2 -29023.621} C_VEL
LIN {X 0,Y 78.157,Z 534.462,A -85,B 0,C 180,E1 -29029.321,E2 -29029.321} C_VEL
LIN {X 0,Y 71.252,Z 540.666,A -85,B 0,C 180,E1 -29037.154,E2 -29037.154} C_VEL
LIN {X 0,Y 66.376,Z 544.742,A -85,B 0,C 180,E1 -29044.95,E2 -29044.95} C_VEL
LIN {X 0,Y 63.575,Z 546.936,A -85,B 0,C 180,E1 -29050.639,E2 -29050.639} C_VEL
LIN {X 0,Y 61.603,Z 548.622,A -85,B 0,C 180,E1 -29056.818,E2 -29056.818} C_VEL
LIN {X 0,Y 59.873,Z 550.79,A -85,B 0,C 180,E1 -29070.007,E2 -29070.007} C_VEL
LIN {X 0,Y 59.934,Z 551.092,A -85,B 0,C 180,E1 -29074.112,E2 -29074.112} C_VEL
LIN {X 0,Y 59.514,Z 551.428,A -85,B 0,C 180,E1 -29077.897,E2 -29077.897} C_VEL
LIN {X 0,Y 57.432,Z 551.926,A -85,B 0,C 180,E1 -29084.19,E2 -29084.19} C_VEL
LIN {X 0,Y 56.036,Z 552.116,A -85,B 0,C 180,E1 -29090.882,E2 -29090.882} C_VEL
LIN {X 0,Y 56.699,Z 551.87,A -85,B 0,C 180,E1 -29094.867,E2 -29094.867} C_VEL
LIN {X 0,Y 61.901,Z 550.32,A -85,B 0,C 180,E1 -29104.597,E2 -29104.597} C_VEL
LIN {X 0,Y 65.757,Z 548.798,A -85,B 0,C 180,E1 -29109.895,E2 -29109.895} C_VEL
LIN {X 0,Y 71.878,Z 545.881,A -85,B 0,C 180,E1 -29116.806,E2 -29116.806} C_VEL
LIN {X 0,Y 79.19,Z 541.706,A -85,B 0,C 180,E1 -29123.018,E2 -29123.018} C_VEL
LIN {X 0,Y 80.853,Z 540.689,A -85,B 0,C 180,E1 -29124.179,E2 -29124.179} C_VEL
LIN {X 0,Y 82.246,Z 539.548,A -85,B 0,C 180,E1 -29125.899,E2 -29125.899} C_VEL
LIN {X 0,Y 67.127,Z 544.955,A -85,B 0,C 180,E1 -29141.692,E2 -29141.692} C_VEL
LIN {X 0,Y 61.802,Z 553.015,A -85,B 0,C 180,E1 -29179.946,E2 -29179.946} C_VEL
LIN {X 0,Y 70.178,Z 556.534,A -85,B 0,C 180,E1 -29196.749,E2 -29196.749} C_VEL
LIN {X 0,Y 63.043,Z 560.523,A -85,B 0,C 180,E1 -29203.554,E2 -29203.554} C_VEL
LIN {X 0,Y 57.097,Z 563.507,A -85,B 0,C 180,E1 -29212.007,E2 -29212.007} C_VEL
LIN {X 0,Y 51.993,Z 566.089,A -85,B 0,C 180,E1 -29226.067,E2 -29226.067} C_VEL
LIN {X 0,Y 50.752,Z 566.869,A -85,B 0,C 180,E1 -29235.768,E2 -29235.768} C_VEL
LIN {X 0,Y 51.349,Z 566.927,A -85,B 0,C 180,E1 -29249.991,E2 -29249.991} C_VEL
LIN {X 0,Y 50.481,Z 565.284,A -85,B 0,C 180,E1 -29262.964,E2 -29262.964} C_VEL
LIN {X 0,Y 52.526,Z 561.939,A -85,B 0,C 180,E1 -29277.914,E2 -29277.914} C_VEL
LIN {X 0,Y 56.517,Z 558.139,A -85,B 0,C 180,E1 -29288.434,E2 -29288.434} C_VEL
LIN {X 0,Y 62.55,Z 552.949,A -85,B 0,C 180,E1 -29297.614,E2 -29297.614} C_VEL
LIN {X 0,Y 69.151,Z 547.056,A -85,B 0,C 180,E1 -29304.384,E2 -29304.384} C_VEL
LIN {X 0,Y 75.832,Z 539.181,A -85,B 0,C 180,E1 -29311.465,E2 -29311.465} C_VEL
LIN {X 0,Y 82.369,Z 531.013,A -85,B 0,C 180,E1 -29316.509,E2 -29316.509} C_VEL
LIN {X 0,Y 89.297,Z 521.253,A -85,B 0,C 180,E1 -29320.796,E2 -29320.796} C_VEL
LIN {X 0,Y 95.892,Z 510.467,A -85,B 0,C 180,E1 -29324.123,E2 -29324.123} C_VEL
LIN {X 0,Y 96.631,Z 509.129,A -85,B 0,C 180,E1 -29324.491,E2 -29324.491} C_VEL
LIN {X 0,Y 97.006,Z 507.849,A -85,B 0,C 180,E1 -29325.31,E2 -29325.31} C_VEL
LIN {X 0,Y 96.813,Z 504.389,A -85,B 0,C 180,E1 -29329.545,E2 -29329.545} C_VEL
LIN {X 0,Y 96.404,Z 500.96,A -85,B 0,C 180,E1 -29335.82,E2 -29335.82} C_VEL
LIN {X 0,Y 96.399,Z 499.23,A -85,B 0,C 180,E1 -29340.001,E2 -29340.001} C_VEL
LIN {X 0,Y 96.381,Z 498.395,A -85,B 0,C 180,E1 -29344.183,E2 -29344.183} C_VEL
LIN {X 0,Y 96.119,Z 498.79,A -85,B 0,C 180,E1 -29348.41,E2 -29348.41} C_VEL
LIN {X 0,Y 95.934,Z 499.875,A -85,B 0,C 180,E1 -29352.697,E2 -29352.697} C_VEL
LIN {X 0,Y 96.003,Z 501.719,A -85,B 0,C 180,E1 -29357.9,E2 -29357.9} C_VEL
LIN {X 0,Y 95.976,Z 503.647,A -85,B 0,C 180,E1 -29361.478,E2 -29361.478} C_VEL
LIN {X 0,Y 95.699,Z 506.896,A -85,B 0,C 180,E1 -29366.145,E2 -29366.145} C_VEL
LIN {X 0,Y 94.891,Z 511.355,A -85,B 0,C 180,E1 -29371.23,E2 -29371.23} C_VEL
LIN {X 0,Y 94.451,Z 512.429,A -85,B 0,C 180,E1 -29372.119,E2 -29372.119} C_VEL
LIN {X 0,Y 86.773,Z 521.873,A -85,B 0,C 180,E1 -29375.921,E2 -29375.921} C_VEL
LIN {X 0,Y 79.006,Z 530.01,A -85,B 0,C 180,E1 -29380.886,E2 -29380.886} C_VEL
LIN {X 0,Y 71.842,Z 536.543,A -85,B 0,C 180,E1 -29386.791,E2 -29386.791} C_VEL
LIN {X 0,Y 65.484,Z 541.75,A -85,B 0,C 180,E1 -29393.832,E2 -29393.832} C_VEL
LIN {X 0,Y 60.093,Z 545.809,A -85,B 0,C 180,E1 -29402.116,E2 -29402.116} C_VEL
LIN {X 0,Y 56.994,Z 547.992,A -85,B 0,C 180,E1 -29408.297,E2 -29408.297} C_VEL
LIN {X 0,Y 53.387,Z 550.932,A -85,B 0,C 180,E1 -29422.444,E2 -29422.444} C_VEL
LIN {X 0,Y 52.913,Z 552.092,A -85,B 0,C 180,E1 -29434.419,E2 -29434.419} C_VEL
LIN {X 0,Y 54.078,Z 552.397,A -85,B 0,C 180,E1 -29445.074,E2 -29445.074} C_VEL
LIN {X 0,Y 56.699,Z 551.87,A -85,B 0,C 180,E1 -29454.867,E2 -29454.867} C_VEL
LIN {X 0,Y 58.546,Z 551.329,A -85,B 0,C 180,E1 -29460.432,E2 -29460.432} C_VEL
LIN {X 0,Y 61.01,Z 550.082,A -85,B 0,C 180,E1 -29469.598,E2 -29469.598} C_VEL
LIN {X 0,Y 63.713,Z 548.616,A -85,B 0,C 180,E1 -29476.378,E2 -29476.378} C_VEL
LIN {X 0,Y 66.752,Z 547.075,A -85,B 0,C 180,E1 -29480.662,E2 -29480.662} C_VEL
LIN {X 0,Y 68.005,Z 546.443,A -85,B 0,C 180,E1 -29481.858,E2 -29481.858} C_VEL
LIN {X 0,Y 71.356,Z 544.751,A -85,B 0,C 180,E1 -29484.552,E2 -29484.552} C_VEL
LIN {X 0,Y 72.3,Z 544.064,A -85,B 0,C 180,E1 -29486.515,E2 -29486.515} C_VEL
LIN {X 0,Y 60.86,Z 547.851,A -85,B 0,C 180,E1 -29499.729,E2 -29499.729} C_VEL
LIN {X 0,Y 54.089,Z 554.384,A -85,B 0,C 180,E1 -29535.06,E2 -29535.06} C_VEL
LIN {X 0,Y 61.152,Z 557.972,A -85,B 0,C 180,E1 -29555.072,E2 -29555.072} C_VEL
LIN {X 0,Y 60.89,Z 558.369,A -85,B 0,C 180,E1 -29556.092,E2 -29556.092} C_VEL
LIN {X 0,Y 55.986,Z 560.68,A -85,B 0,C 180,E1 -29561.122,E2 -29561.122} C_VEL
LIN {X 0,Y 51.653,Z 562.524,A -85,B 0,C 180,E1 -29567.121,E2 -29567.121} C_VEL
LIN {X 0,Y 45.54,Z 565.087,A -85,B 0,C 180,E1 -29582.41,E2 -29582.41} C_VEL
LIN {X 0,Y 43.797,Z 565.886,A -85,B 0,C 180,E1 -29594.316,E2 -29594.316} C_VEL
LIN {X 0,Y 44.199,Z 565.892,A -85,B 0,C 180,E1 -29609.99,E2 -29609.99} C_VEL
LIN {X 0,Y 43.439,Z 564.388,A -85,B 0,C 180,E1 -29623.905,E2 -29623.905} C_VEL
LIN {X 0,Y 46.274,Z 560.852,A -85,B 0,C 180,E1 -29642.1,E2 -29642.1} C_VEL
LIN {X 0,Y 51.072,Z 557.036,A -85,B 0,C 180,E1 -29653.463,E2 -29653.463} C_VEL
LIN {X 0,Y 58.171,Z 551.641,A -85,B 0,C 180,E1 -29663.142,E2 -29663.142} C_VEL
LIN {X 0,Y 63.87,Z 547.058,A -85,B 0,C 180,E1 -29668.501,E2 -29668.501} C_VEL
LIN {X 0,Y 71.808,Z 538.729,A -85,B 0,C 180,E1 -29676.148,E2 -29676.148} C_VEL
LIN {X 0,Y 79.643,Z 529.749,A -85,B 0,C 180,E1 -29681.534,E2 -29681.534} C_VEL
LIN {X 0,Y 87.122,Z 519.955,A -85,B 0,C 180,E1 -29685.449,E2 -29685.449} C_VEL
LIN {X 0,Y 91.956,Z 512.682,A -85,B 0,C 180,E1 -29687.637,E2 -29687.637} C_VEL
LIN {X 0,Y 92.49,Z 511.708,A -85,B 0,C 180,E1 -29688.05,E2 -29688.05} C_VEL
LIN {X 0,Y 92.529,Z 509.403,A -85,B 0,C 180,E1 -29691.264,E2 -29691.264} C_VEL
LIN {X 0,Y 92.428,Z 507.126,A -85,B 0,C 180,E1 -29695.64,E2 -29695.64} C_VEL
LIN {X 0,Y 92.501,Z 505.375,A -85,B 0,C 180,E1 -29700.001,E2 -29700.001} C_VEL
LIN {X 0,Y 92.557,Z 504.419,A -85,B 0,C 180,E1 -29704.356,E2 -29704.356} C_VEL
LIN {X 0,Y 92.17,Z 504.883,A -85,B 0,C 180,E1 -29708.773,E2 -29708.773} C_VEL
LIN {X 0,Y 91.869,Z 506.018,A -85,B 0,C 180,E1 -29713.269,E2 -29713.269} C_VEL
LIN {X 0,Y 91.653,Z 507.644,A -85,B 0,C 180,E1 -29717.863,E2 -29717.863} C_VEL
LIN {X 0,Y 91.26,Z 510.178,A -85,B 0,C 180,E1 -29722.648,E2 -29722.648} C_VEL
LIN {X 0,Y 90.241,Z 514.04,A -85,B 0,C 180,E1 -29727.86,E2 -29727.86} C_VEL
LIN {X 0,Y 89.938,Z 514.875,A -85,B 0,C 180,E1 -29728.762,E2 -29728.762} C_VEL
LIN {X 0,Y 82.856,Z 523.04,A -85,B 0,C 180,E1 -29731.993,E2 -29731.993} C_VEL
LIN {X 0,Y 74.604,Z 531.139,A -85,B 0,C 180,E1 -29736.811,E2 -29736.811} C_VEL
LIN {X 0,Y 66.913,Z 537.647,A -85,B 0,C 180,E1 -29742.684,E2 -29742.684} C_VEL
LIN {X 0,Y 59.974,Z 542.834,A -85,B 0,C 180,E1 -29749.881,E2 -29749.881} C_VEL
LIN {X 0,Y 53.989,Z 546.877,A -85,B 0,C 180,E1 -29758.631,E2 -29758.631} C_VEL
LIN {X 0,Y 50.554,Z 549.043,A -85,B 0,C 180,E1 -29765.361,E2 -29765.361} C_VEL
LIN {X 0,Y 46.43,Z 551.966,A -85,B 0,C 180,E1 -29781.304,E2 -29781.304} C_VEL
LIN {X 0,Y 45.816,Z 552.841,A -85,B 0,C 180,E1 -29790.01,E2 -29790.01} C_VEL
LIN {X 0,Y 46.201,Z 553.302,A -85,B 0,C 180,E1 -29798.759,E2 -29798.759} C_VEL
LIN {X 0,Y 49.281,Z 553.131,A -85,B 0,C 180,E1 -29815.339,E2 -29815.339} C_VEL
LIN {X 0,Y 52.393,Z 552.434,A -85,B 0,C 180,E1 -29822.459,E2 -29822.459} C_VEL
LIN {X 0,Y 56.256,Z 551.286,A -85,B 0,C 180,E1 -29828.666,E2 -29828.666} C_VEL
LIN {X 0,Y 60.529,Z 549.755,A -85,B 0,C 180,E1 -29834.169,E2 -29834.169} C_VEL
LIN {X 0,Y 68.005,Z 546.443,A -85,B 0,C 180,E1 -29841.858,E2 -29841.858} C_VEL
LIN {X 0,Y 66.93,Z 546.814,A -85,B 0,C 180,E1 -29842.125,E2 -29842.125} C_VEL
LIN {X 0,Y 61.606,Z 548.858,A -85,B 0,C 180,E1 -29840.355,E2 -29840.355} C_VEL
LIN {X 0,Y 55.632,Z 550.918,A -85,B 0,C 180,E1 -29836.491,E2 -29836.491} C_VEL
LIN {X 0,Y 51.227,Z 552.238,A -85,B 0,C 180,E1 -29832.609,E2 -29832.609} C_VEL
LIN {X 0,Y 45.531,Z 553.637,A -85,B 0,C 180,E1 -29824.922,E2 -29824.922} C_VEL
LIN {X 0,Y 44.004,Z 553.913,A -85,B 0,C 180,E1 -29821.775,E2 -29821.775} C_VEL
LIN {X 0,Y 40.664,Z 554.397,A -85,B 0,C 180,E1 -29810.233,E2 -29810.233} C_VEL
LIN {X 0,Y 39.268,Z 554.311,A -85,B 0,C 180,E1 -29800.321,E2 -29800.321} C_VEL
LIN {X 0,Y 38.788,Z 553.867,A -85,B 0,C 180,E1 -29790.011,E2 -29790.011} C_VEL
LIN {X 0,Y 41.362,Z 551.748,A -85,B 0,C 180,E1 -29770.145,E2 -29770.145} C_VEL
LIN {X 0,Y 46.165,Z 549.052,A -85,B 0,C 180,E1 -29757.815,E2 -29757.815} C_VEL
LIN {X 0,Y 52.452,Z 545.377,A -85,B 0,C 180,E1 -29747.949,E2 -29747.949} C_VEL
LIN {X 0,Y 59.77,Z 540.612,A -85,B 0,C 180,E1 -29740.168,E2 -29740.168} C_VEL
LIN {X 0,Y 67.765,Z 534.624,A -85,B 0,C 180,E1 -29733.945,E2 -29733.945} C_VEL
LIN {X 0,Y 76.406,Z 527.087,A -85,B 0,C 180,E1 -29729.106,E2 -29729.106} C_VEL
LIN {X 0,Y 84.085,Z 519.169,A -85,B 0,C 180,E1 -29725.729,E2 -29725.729} C_VEL
LIN {X 0,Y 85.446,Z 517.641,A -85,B 0,C 180,E1 -29725.223,E2 -29725.223} C_VEL
LIN {X 0,Y 86.282,Z 515.534,A -85,B 0,C 180,E1 -29722.119,E2 -29722.119} C_VEL
LIN {X 0,Y 86.904,Z 513.77,A -85,B 0,C 180,E1 -29718.875,E2 -29718.875} C_VEL
LIN {X 0,Y 87.356,Z 511.966,A -85,B 0,C 180,E1 -29713.968,E2 -29713.968} C_VEL
LIN {X 0,Y 87.869,Z 510.782,A -85,B 0,C 180,E1 -29709.206,E2 -29709.206} C_VEL
LIN {X 0,Y 88.396,Z 510.214,A -85,B 0,C 180,E1 -29704.561,E2 -29704.561} C_VEL
LIN {X 0,Y 88.253,Z 511.272,A -85,B 0,C 180,E1 -29700.001,E2 -29700.001} C_VEL
LIN {X 0,Y 88.088,Z 513.096,A -85,B 0,C 180,E1 -29695.425,E2 -29695.425} C_VEL
LIN {X 0,Y 87.999,Z 515.148,A -85,B 0,C 180,E1 -29691.526,E2 -29691.526} C_VEL
LIN {X 0,Y 86.303,Z 517.609,A -85,B 0,C 180,E1 -29690.628,E2 -29690.628} C_VEL
LIN {X 0,Y 77.589,Z 528.497,A -85,B 0,C 180,E1 -29686.811,E2 -29686.811} C_VEL
LIN {X 0,Y 68.552,Z 538.038,A -85,B 0,C 180,E1 -29681.528,E2 -29681.528} C_VEL
LIN {X 0,Y 60.282,Z 545.861,A -85,B 0,C 180,E1 -29674.609,E2 -29674.609} C_VEL
LIN {X 0,Y 56.202,Z 549.085,A -85,B 0,C 180,E1 -29671.068,E2 -29671.068} C_VEL
LIN {X 0,Y 48.418,Z 554.426,A -85,B 0,C 180,E1 -29662.956,E2 -29662.956} C_VEL
LIN {X 0,Y 42.021,Z 558.611,A -85,B 0,C 180,E1 -29651.975,E2 -29651.975} C_VEL
LIN {X 0,Y 36.968,Z 562.587,A -85,B 0,C 180,E1 -29632.334,E2 -29632.334} C_VEL
LIN {X 0,Y 36.348,Z 563.954,A -85,B 0,C 180,E1 -29621.136,E2 -29621.136} C_VEL
LIN {X 0,Y 37.047,Z 564.858,A -85,B 0,C 180,E1 -29609.988,E2 -29609.988} C_VEL
LIN {X 0,Y 36.851,Z 564.905,A -85,B 0,C 180,E1 -29592.462,E2 -29592.462} C_VEL
LIN {X 0,Y 39.324,Z 564.082,A -85,B 0,C 180,E1 -29577.564,E2 -29577.564} C_VEL
LIN {X 0,Y 46.674,Z 561.543,A -85,B 0,C 180,E1 -29561.146,E2 -29561.146} C_VEL
LIN {X 0,Y 51.573,Z 559.708,A -85,B 0,C 180,E1 -29555.138,E2 -29555.138} C_VEL
LIN {X 0,Y 52.091,Z 559.012,A -85,B 0,C 180,E1 -29552.659,E2 -29552.659} C_VEL
LIN {X 0,Y 47.313,Z 554.169,A -85,B 0,C 180,E1 -29519.998,E2 -29519.998} C_VEL
LIN {X 0,Y 58.603,Z 549.042,A -85,B 0,C 180,E1 -29491.332,E2 -29491.332} C_VEL
LIN {X 0,Y 62.767,Z 547.896,A -85,B 0,C 180,E1 -29485.953,E2 -29485.953} C_VEL
LIN {X 0,Y 55.699,Z 550.712,A -85,B 0,C 180,E1 -29479.217,E2 -29479.217} C_VEL
LIN {X 0,Y 50.956,Z 552.252,A -85,B 0,C 180,E1 -29473.611,E2 -29473.611} C_VEL
LIN {X 0,Y 44.004,Z 553.913,A -85,B 0,C 180,E1 -29461.775,E2 -29461.775} C_VEL
LIN {X 0,Y 40.895,Z 554.46,A -85,B 0,C 180,E1 -29454.993,E2 -29454.993} C_VEL
LIN {X 0,Y 35.618,Z 554.98,A -85,B 0,C 180,E1 -29442.349,E2 -29442.349} C_VEL
LIN {X 0,Y 32.775,Z 554.809,A -85,B 0,C 180,E1 -29429.862,E2 -29429.862} C_VEL
LIN {X 0,Y 32.453,Z 554.198,A -85,B 0,C 180,E1 -29419.5,E2 -29419.5} C_VEL
LIN {X 0,Y 32.804,Z 553.884,A -85,B 0,C 180,E1 -29416.128,E2 -29416.128} C_VEL
LIN {X 0,Y 38.266,Z 551.142,A -85,B 0,C 180,E1 -29396.579,E2 -29396.579} C_VEL
LIN {X 0,Y 44.999,Z 547.805,A -85,B 0,C 180,E1 -29385.36,E2 -29385.36} C_VEL
LIN {X 0,Y 52.721,Z 543.45,A -85,B 0,C 180,E1 -29376.9,E2 -29376.9} C_VEL
LIN {X 0,Y 62.673,Z 536.808,A -85,B 0,C 180,E1 -29369.664,E2 -29369.664} C_VEL
LIN {X 0,Y 71.719,Z 529.597,A -85,B 0,C 180,E1 -29364.997,E2 -29364.997} C_VEL
LIN {X 0,Y 79.669,Z 522.069,A -85,B 0,C 180,E1 -29361.831,E2 -29361.831} C_VEL
LIN {X 0,Y 81.134,Z 520.493,A -85,B 0,C 180,E1 -29361.226,E2 -29361.226} C_VEL
LIN {X 0,Y 81.719,Z 519.312,A -85,B 0,C 180,E1 -29358.929,E2 -29358.929} C_VEL
LIN {X 0,Y 82.436,Z 517.749,A -85,B 0,C 180,E1 -29354.82,E2 -29354.82} C_VEL
LIN {X 0,Y 83.178,Z 516.456,A -85,B 0,C 180,E1 -29349.73,E2 -29349.73} C_VEL
LIN {X 0,Y 83.888,Z 515.818,A -85,B 0,C 180,E1 -29344.807,E2 -29344.807} C_VEL
LIN {X 0,Y 83.667,Z 516.948,A -85,B 0,C 180,E1 -29340.001,E2 -29340.001} C_VEL
LIN {X 0,Y 83.383,Z 518.845,A -85,B 0,C 180,E1 -29335.166,E2 -29335.166} C_VEL
LIN {X 0,Y 80.873,Z 521.984,A -85,B 0,C 180,E1 -29334.025,E2 -29334.025} C_VEL
LIN {X 0,Y 72.944,Z 530.671,A -85,B 0,C 180,E1 -29330.911,E2 -29330.911} C_VEL
LIN {X 0,Y 63.416,Z 539.616,A -85,B 0,C 180,E1 -29325.832,E2 -29325.832} C_VEL
LIN {X 0,Y 54.583,Z 546.899,A -85,B 0,C 180,E1 -29318.961,E2 -29318.961} C_VEL
LIN {X 0,Y 44.458,Z 553.322,A -85,B 0,C 180,E1 -29310.374,E2 -29310.374} C_VEL
LIN {X 0,Y 36.977,Z 557.523,A -85,B 0,C 180,E1 -29299.469,E2 -29299.469} C_VEL
LIN {X 0,Y 33.084,Z 559.728,A -85,B 0,C 180,E1 -29289.571,E2 -29289.571} C_VEL
LIN {X 0,Y 29.32,Z 562.9,A -85,B 0,C 180,E1 -29263.853,E2 -29263.853} C_VEL
LIN {X 0,Y 29.893,Z 563.823,A -85,B 0,C 180,E1 -29249.985,E2 -29249.985} C_VEL
LIN {X 0,Y 29.988,Z 563.922,A -85,B 0,C 180,E1 -29229.617,E2 -29229.617} C_VEL
LIN {X 0,Y 33.51,Z 563.08,A -85,B 0,C 180,E1 -29210.993,E2 -29210.993} C_VEL
LIN {X 0,Y 42.323,Z 560.562,A -85,B 0,C 180,E1 -29193.854,E2 -29193.854} C_VEL
LIN {X 0,Y 43.284,Z 560.272,A -85,B 0,C 180,E1 -29192.717,E2 -29192.717} C_VEL
LIN {X 0,Y 43.183,Z 559.68,A -85,B 0,C 180,E1 -29189.223,E2 -29189.223} C_VEL
LIN {X 0,Y 43.982,Z 553.965,A -85,B 0,C 180,E1 -29143.518,E2 -29143.518} C_VEL
LIN {X 0,Y 52.656,Z 551.224,A -85,B 0,C 180,E1 -29127.73,E2 -29127.73} C_VEL
LIN {X 0,Y 51.381,Z 551.669,A -85,B 0,C 180,E1 -29125.168,E2 -29125.168} C_VEL
LIN {X 0,Y 46.121,Z 553.217,A -85,B 0,C 180,E1 -29119.647,E2 -29119.647} C_VEL
LIN {X 0,Y 38.077,Z 554.925,A -85,B 0,C 180,E1 -29107.059,E2 -29107.059} C_VEL
LIN {X 0,Y 34.153,Z 555.398,A -85,B 0,C 180,E1 -29094.316,E2 -29094.316} C_VEL
LIN {X 0,Y 32.377,Z 555.32,A -85,B 0,C 180,E1 -29082.551,E2 -29082.551} C_VEL
LIN {X 0,Y 31.76,Z 554.89,A -85,B 0,C 180,E1 -29070.014,E2 -29070.014} C_VEL
LIN {X 0,Y 32.804,Z 553.884,A -85,B 0,C 180,E1 -29056.128,E2 -29056.128} C_VEL
LIN {X 0,Y 34.088,Z 552.981,A -85,B 0,C 180,E1 -29046.376,E2 -29046.376} C_VEL
LIN {X 0,Y 36.603,Z 551.12,A -85,B 0,C 180,E1 -29031.048,E2 -29031.048} C_VEL
LIN {X 0,Y 40.01,Z 549.149,A -85,B 0,C 180,E1 -29020.67,E2 -29020.67} C_VEL
LIN {X 0,Y 43.7,Z 547.234,A -85,B 0,C 180,E1 -29014.87,E2 -29014.87} C_VEL
LIN {X 0,Y 45.151,Z 546.482,A -85,B 0,C 180,E1 -29013.412,E2 -29013.412} C_VEL
LIN {X 0,Y 54.885,Z 540.964,A -85,B 0,C 180,E1 -29006.338,E2 -29006.338} C_VEL
LIN {X 0,Y 64.245,Z 534.528,A -85,B 0,C 180,E1 -29001.609,E2 -29001.609} C_VEL
LIN {X 0,Y 73.9,Z 526.523,A -85,B 0,C 180,E1 -28998.028,E2 -28998.028} C_VEL
LIN {X 0,Y 75.22,Z 525.274,A -85,B 0,C 180,E1 -28997.633,E2 -28997.633} C_VEL
LIN {X 0,Y 77.017,Z 523.385,A -85,B 0,C 180,E1 -28995.889,E2 -28995.889} C_VEL
LIN {X 0,Y 78.315,Z 521.666,A -85,B 0,C 180,E1 -28989.239,E2 -28989.239} C_VEL
LIN {X 0,Y 79.033,Z 521.184,A -85,B 0,C 180,E1 -28985.103,E2 -28985.103} C_VEL
LIN {X 0,Y 78.744,Z 522.343,A -85,B 0,C 180,E1 -28980.001,E2 -28980.001} C_VEL
LIN {X 0,Y 77.327,Z 524.127,A -85,B 0,C 180,E1 -28978.485,E2 -28978.485} C_VEL
LIN {X 0,Y 68.745,Z 532.6,A -85,B 0,C 180,E1 -28975.548,E2 -28975.548} C_VEL
LIN {X 0,Y 58.715,Z 541.028,A -85,B 0,C 180,E1 -28970.881,E2 -28970.881} C_VEL
LIN {X 0,Y 50.795,Z 546.802,A -85,B 0,C 180,E1 -28965.549,E2 -28965.549} C_VEL
LIN {X 0,Y 41.382,Z 552.217,A -85,B 0,C 180,E1 -28959.048,E2 -28959.048} C_VEL
LIN {X 0,Y 32.756,Z 556.436,A -85,B 0,C 180,E1 -28949.091,E2 -28949.091} C_VEL
LIN {X 0,Y 27.909,Z 558.651,A -85,B 0,C 180,E1 -28939.04,E2 -28939.04} C_VEL
LIN {X 0,Y 22.389,Z 561.843,A -85,B 0,C 180,E1 -28908.274,E2 -28908.274} C_VEL
LIN {X 0,Y 22.702,Z 562.782,A -85,B 0,C 180,E1 -28889.981,E2 -28889.981} C_VEL
LIN {X 0,Y 23.265,Z 562.929,A -85,B 0,C 180,E1 -28864.98,E2 -28864.98} C_VEL
LIN {X 0,Y 28.303,Z 562.073,A -85,B 0,C 180,E1 -28841.823,E2 -28841.823} C_VEL
LIN {X 0,Y 33.186,Z 561.021,A -85,B 0,C 180,E1 -28832.079,E2 -28832.079} C_VEL
LIN {X 0,Y 35.053,Z 560.261,A -85,B 0,C 180,E1 -28826.864,E2 -28826.864} C_VEL
LIN {X 0,Y 42.089,Z 554.156,A -85,B 0,C 180,E1 -28769.935,E2 -28769.935} C_VEL
LIN {X 0,Y 41.912,Z 554.183,A -85,B 0,C 180,E1 -28766.992,E2 -28766.992} C_VEL
LIN {X 0,Y 36.398,Z 555.371,A -85,B 0,C 180,E1 -28760.584,E2 -28760.584} C_VEL
